--- program P_fl_2 (robot KUKA KR 16 2) ---
  Suave(1)
  Establecer velocidad (1000.0 mm/s)
  Est. Ref.: Frame 2
  Est. herr: Plumon_ensamble
  Mostrar Plumon_ensamble
  MoveJ 1 to (150.76, 185.35, 20) mm, rotated rx -180 ry 0 rz -39.83 deg; joints [47.982, -66.548, 70.781, -0.863, 85.768, 48.043]
  MoveL 2 to (150.76, 185.35, 20) mm, rotated rx -180 ry 0 rz -39.83 deg; joints [47.982, -66.548, 70.781, -0.863, 85.768, 48.043]
  MoveL 3 to (150.76, 185.35, 0) mm, rotated rx -180 ry 0 rz -39.83 deg; joints [47.968, -66.304, 72.161, -0.865, 84.143, 48.053]
  MoveL 4 to (150.76, 185.35, 0) mm, rotated rx -180 ry 0 rz -39.83 deg; joints [47.968, -66.304, 72.161, -0.865, 84.143, 48.053]
  Establecer velocidad (50.0 mm/s)
  MoveL 5 to (150.39, 185.32, 0) mm, rotated rx 180 ry 0 rz -39.83 deg; joints [47.95, -66.305, 72.163, -0.865, 84.143, 48.036]
  MoveL 6 to (150.03, 185.29, 0) mm, rotated rx 180 ry 0 rz -39.83 deg; joints [47.933, -66.307, 72.164, -0.865, 84.143, 48.018]
  MoveL 7 to (149.66, 185.26, 0) mm, rotated rx 180 ry 0 rz -39.83 deg; joints [47.915, -66.308, 72.165, -0.865, 84.142, 48]
  MoveL 8 to (149.29, 185.23, 0) mm, rotated rx 180 ry 0 rz -39.83 deg; joints [47.898, -66.309, 72.166, -0.865, 84.142, 47.983]
  MoveL 9 to (148.29, 185.2, 0) mm, rotated rx 180 ry 0 rz -39.83 deg; joints [47.85, -66.309, 72.165, -0.865, 84.143, 47.935]
  MoveL 10 to (147.29, 185.19, 0) mm, rotated rx 180 ry 0 rz -39.83 deg; joints [47.802, -66.306, 72.159, -0.865, 84.144, 47.887]
  MoveL 11 to (146.29, 185.21, 0) mm, rotated rx -180 ry 0 rz -39.83 deg; joints [47.754, -66.301, 72.151, -0.865, 84.147, 47.839]
  MoveL 12 to (145.28, 185.23, 0) mm, rotated rx -180 ry 0 rz -39.83 deg; joints [47.706, -66.295, 72.142, -0.865, 84.15, 47.791]
  MoveL 13 to (144.05, 185.27, 0) mm, rotated rx 180 ry 0 rz -39.83 deg; joints [47.647, -66.288, 72.129, -0.865, 84.154, 47.732]
  MoveL 14 to (142.82, 185.33, 0) mm, rotated rx -180 ry 0 rz -39.83 deg; joints [47.588, -66.278, 72.115, -0.865, 84.158, 47.673]
  MoveL 15 to (141.59, 185.42, 0) mm, rotated rx 180 ry 0 rz -39.83 deg; joints [47.53, -66.266, 72.096, -0.865, 84.164, 47.614]
  MoveL 16 to (140.37, 185.55, 0) mm, rotated rx -180 ry 0 rz -39.83 deg; joints [47.472, -66.25, 72.072, -0.865, 84.172, 47.556]
  MoveL 17 to (139.51, 185.68, 0) mm, rotated rx 180 ry 0 rz -39.83 deg; joints [47.431, -66.235, 72.05, -0.865, 84.178, 47.515]
  MoveL 18 to (138.64, 185.84, 0) mm, rotated rx 180 ry 0 rz -39.83 deg; joints [47.39, -66.219, 72.025, -0.865, 84.186, 47.474]
  MoveL 19 to (137.78, 186.01, 0) mm, rotated rx 180 ry 0 rz -39.83 deg; joints [47.349, -66.2, 71.997, -0.865, 84.194, 47.433]
  MoveL 20 to (136.93, 186.2, 0) mm, rotated rx 180 ry 0 rz -39.83 deg; joints [47.308, -66.18, 71.968, -0.865, 84.202, 47.393]
  MoveL 21 to (135.83, 186.46, 0) mm, rotated rx 180 ry 0 rz -39.83 deg; joints [47.257, -66.153, 71.929, -0.865, 84.214, 47.34]
  MoveL 22 to (134.73, 186.74, 0) mm, rotated rx 180 ry 0 rz -39.83 deg; joints [47.205, -66.125, 71.887, -0.865, 84.227, 47.289]
  MoveL 23 to (133.64, 187.03, 0) mm, rotated rx -180 ry 0 rz -39.83 deg; joints [47.154, -66.095, 71.843, -0.865, 84.24, 47.237]
  MoveL 24 to (132.56, 187.35, 0) mm, rotated rx 180 ry 0 rz -39.83 deg; joints [47.103, -66.063, 71.796, -0.865, 84.254, 47.186]
  MoveL 25 to (131.68, 187.63, 0) mm, rotated rx 180 ry 0 rz -39.83 deg; joints [47.062, -66.035, 71.756, -0.865, 84.266, 47.145]
  MoveL 26 to (130.81, 187.93, 0) mm, rotated rx -180 ry 0 rz -39.83 deg; joints [47.021, -66.005, 71.712, -0.865, 84.279, 47.104]
  MoveL 27 to (129.95, 188.26, 0) mm, rotated rx 180 ry 0 rz -39.83 deg; joints [46.981, -65.972, 71.665, -0.865, 84.293, 47.063]
  MoveL 28 to (129.1, 188.62, 0) mm, rotated rx -180 ry 0 rz -39.83 deg; joints [46.941, -65.937, 71.614, -0.865, 84.308, 47.024]
  MoveL 29 to (128.38, 188.97, 0) mm, rotated rx 180 ry 0 rz -39.83 deg; joints [46.908, -65.904, 71.566, -0.865, 84.322, 46.99]
  MoveL 30 to (127.67, 189.34, 0) mm, rotated rx 180 ry 0 rz -39.83 deg; joints [46.875, -65.868, 71.515, -0.865, 84.338, 46.957]
  MoveL 31 to (126.97, 189.74, 0) mm, rotated rx 180 ry 0 rz -39.83 deg; joints [46.843, -65.83, 71.46, -0.865, 84.354, 46.925]
  MoveL 32 to (126.29, 190.17, 0) mm, rotated rx -180 ry 0 rz -39.83 deg; joints [46.812, -65.79, 71.401, -0.865, 84.371, 46.893]
  MoveL 33 to (125.71, 190.58, 0) mm, rotated rx 180 ry 0 rz -39.83 deg; joints [46.785, -65.752, 71.347, -0.865, 84.388, 46.866]
  MoveL 34 to (125.14, 191, 0) mm, rotated rx -180 ry 0 rz -39.83 deg; joints [46.76, -65.713, 71.29, -0.865, 84.405, 46.84]
  MoveL 35 to (124.6, 191.45, 0) mm, rotated rx -180 ry 0 rz -39.83 deg; joints [46.735, -65.671, 71.23, -0.865, 84.422, 46.816]
  MoveL 36 to (124.08, 191.93, 0) mm, rotated rx -180 ry 0 rz -39.83 deg; joints [46.712, -65.627, 71.167, -0.864, 84.441, 46.792]
  MoveL 37 to (123.59, 192.43, 0) mm, rotated rx 180 ry 0 rz -39.83 deg; joints [46.69, -65.582, 71.102, -0.864, 84.461, 46.77]
  MoveL 38 to (123.13, 192.95, 0) mm, rotated rx 180 ry 0 rz -39.83 deg; joints [46.669, -65.534, 71.034, -0.864, 84.481, 46.749]
  MoveL 39 to (122.67, 193.48, 0) mm, rotated rx -180 ry 0 rz -39.83 deg; joints [46.649, -65.486, 70.964, -0.864, 84.502, 46.729]
  MoveL 40 to (122.23, 194.03, 0) mm, rotated rx -180 ry 0 rz -39.83 deg; joints [46.63, -65.436, 70.893, -0.864, 84.523, 46.709]
  MoveL 41 to (121.75, 194.65, 0) mm, rotated rx 180 ry 0 rz -39.83 deg; joints [46.609, -65.38, 70.812, -0.864, 84.548, 46.688]
  MoveL 42 to (121.29, 195.28, 0) mm, rotated rx -180 ry 0 rz -39.83 deg; joints [46.589, -65.323, 70.73, -0.864, 84.572, 46.667]
  MoveL 43 to (120.86, 195.94, 0) mm, rotated rx 180 ry 0 rz -39.83 deg; joints [46.571, -65.264, 70.645, -0.864, 84.598, 46.649]
  MoveL 44 to (120.5, 196.62, 0) mm, rotated rx -180 ry 0 rz -39.83 deg; joints [46.556, -65.203, 70.558, -0.864, 84.624, 46.633]
  MoveL 45 to (120.13, 197.53, 0) mm, rotated rx 180 ry 0 rz -39.83 deg; joints [46.541, -65.121, 70.441, -0.864, 84.66, 46.618]
  MoveL 46 to (119.85, 198.49, 0) mm, rotated rx 180 ry 0 rz -39.83 deg; joints [46.531, -65.037, 70.32, -0.864, 84.696, 46.607]
  MoveL 47 to (119.64, 199.47, 0) mm, rotated rx 180 ry 0 rz -39.83 deg; joints [46.523, -64.95, 70.195, -0.864, 84.734, 46.599]
  MoveL 48 to (119.45, 200.46, 0) mm, rotated rx 180 ry 0 rz -39.83 deg; joints [46.518, -64.863, 70.07, -0.864, 84.772, 46.593]
  Establecer velocidad (1000.0 mm/s)
  MoveL 49 to (119.45, 200.46, 0) mm, rotated rx 180 ry 0 rz -39.83 deg; joints [46.518, -64.863, 70.07, -0.864, 84.772, 46.593]
  MoveL 50 to (119.45, 200.46, 20) mm, rotated rx 180 ry 0 rz -39.83 deg; joints [46.532, -65.091, 68.674, -0.862, 86.395, 46.583]
  Establecer velocidad (1000.0 mm/s)
  MoveL 51 to (146.94, 188.19, 20) mm, rotated rx 180 ry 0 rz -39.83 deg; joints [47.806, -66.288, 70.409, -0.863, 85.877, 47.864]
  MoveL 52 to (146.94, 188.19, 0) mm, rotated rx 180 ry 0 rz -39.83 deg; joints [47.791, -66.046, 71.792, -0.865, 84.252, 47.875]
  MoveL 53 to (146.94, 188.19, 0) mm, rotated rx 180 ry 0 rz -39.83 deg; joints [47.791, -66.046, 71.792, -0.865, 84.252, 47.875]
  Establecer velocidad (50.0 mm/s)
  MoveL 54 to (147.05, 187.92, 0) mm, rotated rx -180 ry 0 rz -39.83 deg; joints [47.796, -66.07, 71.826, -0.865, 84.242, 47.879]
  MoveL 55 to (147.17, 187.65, 0) mm, rotated rx 180 ry 0 rz -39.83 deg; joints [47.801, -66.094, 71.86, -0.865, 84.232, 47.885]
  MoveL 56 to (147.31, 187.4, 0) mm, rotated rx 180 ry 0 rz -39.83 deg; joints [47.807, -66.116, 71.891, -0.865, 84.223, 47.891]
  MoveL 57 to (147.47, 187.17, 0) mm, rotated rx 180 ry 0 rz -39.83 deg; joints [47.814, -66.136, 71.92, -0.865, 84.215, 47.898]
  MoveL 58 to (147.77, 186.91, 0) mm, rotated rx 180 ry 0 rz -39.83 deg; joints [47.828, -66.159, 71.953, -0.865, 84.205, 47.912]
  MoveL 59 to (148.12, 186.7, 0) mm, rotated rx 180 ry 0 rz -39.83 deg; joints [47.844, -66.179, 71.981, -0.865, 84.197, 47.929]
  MoveL 60 to (148.5, 186.52, 0) mm, rotated rx 180 ry 0 rz -39.83 deg; joints [47.862, -66.195, 72.005, -0.865, 84.189, 47.946]
  MoveL 61 to (148.88, 186.35, 0) mm, rotated rx -180 ry 0 rz -39.83 deg; joints [47.88, -66.211, 72.028, -0.865, 84.183, 47.965]
  MoveL 62 to (149.37, 186.12, 0) mm, rotated rx 180 ry 0 rz -39.83 deg; joints [47.903, -66.233, 72.059, -0.865, 84.173, 47.988]
  MoveL 63 to (149.85, 185.87, 0) mm, rotated rx 180 ry 0 rz -39.83 deg; joints [47.925, -66.256, 72.092, -0.865, 84.164, 48.01]
  MoveL 64 to (150.3, 185.61, 0) mm, rotated rx 180 ry 0 rz -39.83 deg; joints [47.947, -66.28, 72.126, -0.865, 84.154, 48.032]
  MoveL 65 to (150.76, 185.35, 0) mm, rotated rx -180 ry 0 rz -39.83 deg; joints [47.968, -66.304, 72.161, -0.865, 84.143, 48.053]
  Establecer velocidad (1000.0 mm/s)
  MoveL 66 to (150.76, 185.35, 0) mm, rotated rx -180 ry 0 rz -39.83 deg; joints [47.968, -66.304, 72.161, -0.865, 84.143, 48.053]
  MoveL 67 to (150.76, 185.35, 20) mm, rotated rx -180 ry 0 rz -39.83 deg; joints [47.982, -66.548, 70.781, -0.863, 85.768, 48.043]
  Establecer velocidad (1000.0 mm/s)
  MoveL 68 to (146.94, 188.19, 20) mm, rotated rx 180 ry 0 rz -39.83 deg; joints [47.806, -66.288, 70.409, -0.863, 85.877, 47.864]
  MoveL 69 to (146.94, 188.19, 0) mm, rotated rx 180 ry 0 rz -39.83 deg; joints [47.791, -66.046, 71.792, -0.865, 84.252, 47.875]
  MoveL 70 to (146.94, 188.19, 0) mm, rotated rx 180 ry 0 rz -39.83 deg; joints [47.791, -66.046, 71.792, -0.865, 84.252, 47.875]
  Establecer velocidad (50.0 mm/s)
  MoveL 71 to (147.49, 188.32, 0) mm, rotated rx -180 ry 0 rz -39.83 deg; joints [47.817, -66.037, 71.779, -0.865, 84.256, 47.901]
  MoveL 72 to (148.03, 188.44, 0) mm, rotated rx -180 ry 0 rz -39.83 deg; joints [47.844, -66.029, 71.768, -0.865, 84.259, 47.927]
  MoveL 73 to (148.58, 188.53, 0) mm, rotated rx -180 ry 0 rz -39.83 deg; joints [47.87, -66.022, 71.76, -0.865, 84.261, 47.953]
  MoveL 74 to (149.12, 188.6, 0) mm, rotated rx 180 ry 0 rz -39.83 deg; joints [47.896, -66.018, 71.755, -0.865, 84.263, 47.979]
  MoveL 75 to (149.7, 188.63, 0) mm, rotated rx 180 ry 0 rz -39.83 deg; joints [47.923, -66.018, 71.755, -0.865, 84.262, 48.007]
  MoveL 76 to (150.27, 188.63, 0) mm, rotated rx -180 ry 0 rz -39.83 deg; joints [47.951, -66.019, 71.758, -0.865, 84.261, 48.034]
  MoveL 77 to (150.85, 188.62, 0) mm, rotated rx 180 ry 0 rz -39.83 deg; joints [47.978, -66.022, 71.762, -0.865, 84.26, 48.062]
  MoveL 78 to (151.43, 188.62, 0) mm, rotated rx 180 ry 0 rz -39.83 deg; joints [48.006, -66.024, 71.766, -0.865, 84.259, 48.089]
  MoveL 79 to (152.23, 188.66, 0) mm, rotated rx 180 ry 0 rz -39.83 deg; joints [48.044, -66.023, 71.766, -0.865, 84.259, 48.128]
  MoveL 80 to (153.02, 188.73, 0) mm, rotated rx 180 ry 0 rz -39.83 deg; joints [48.082, -66.019, 71.761, -0.865, 84.26, 48.166]
  MoveL 81 to (153.81, 188.83, 0) mm, rotated rx 180 ry 0 rz -39.83 deg; joints [48.12, -66.012, 71.753, -0.865, 84.262, 48.204]
  MoveL 82 to (154.6, 188.96, 0) mm, rotated rx 180 ry 0 rz -39.83 deg; joints [48.158, -66.004, 71.742, -0.865, 84.265, 48.241]
  MoveL 83 to (155.12, 189.06, 0) mm, rotated rx 180 ry 0 rz -39.83 deg; joints [48.183, -65.997, 71.733, -0.865, 84.268, 48.266]
  MoveL 84 to (155.65, 189.15, 0) mm, rotated rx 180 ry 0 rz -39.83 deg; joints [48.208, -65.99, 71.723, -0.865, 84.271, 48.291]
  MoveL 85 to (156.18, 189.25, 0) mm, rotated rx 180 ry 0 rz -39.83 deg; joints [48.234, -65.983, 71.714, -0.865, 84.273, 48.317]
  MoveL 86 to (156.72, 189.34, 0) mm, rotated rx 180 ry 0 rz -39.83 deg; joints [48.26, -65.976, 71.706, -0.865, 84.276, 48.343]
  MoveL 87 to (157.41, 189.46, 0) mm, rotated rx 180 ry 0 rz -39.83 deg; joints [48.293, -65.969, 71.696, -0.865, 84.278, 48.376]
  MoveL 88 to (158.09, 189.6, 0) mm, rotated rx 180 ry 0 rz -39.83 deg; joints [48.326, -65.958, 71.682, -0.865, 84.282, 48.409]
  MoveL 89 to (158.73, 189.82, 0) mm, rotated rx 180 ry 0 rz -39.83 deg; joints [48.356, -65.941, 71.658, -0.865, 84.289, 48.439]
  MoveL 90 to (159.28, 190.16, 0) mm, rotated rx 180 ry 0 rz -39.83 deg; joints [48.383, -65.913, 71.619, -0.865, 84.301, 48.466]
  MoveL 91 to (159.48, 190.35, 0) mm, rotated rx 180 ry 0 rz -39.83 deg; joints [48.393, -65.897, 71.597, -0.865, 84.307, 48.475]
  MoveL 92 to (159.66, 190.56, 0) mm, rotated rx 180 ry 0 rz -39.83 deg; joints [48.402, -65.879, 71.572, -0.865, 84.314, 48.484]
  MoveL 93 to (159.83, 190.78, 0) mm, rotated rx 180 ry 0 rz -39.83 deg; joints [48.41, -65.86, 71.545, -0.865, 84.322, 48.493]
  MoveL 94 to (160, 191.02, 0) mm, rotated rx 180 ry 0 rz -39.83 deg; joints [48.419, -65.84, 71.517, -0.865, 84.331, 48.501]
  MoveL 95 to (160, 191.02, 0) mm, rotated rx 180 ry 0 rz -39.83 deg; joints [48.419, -65.84, 71.517, -0.865, 84.331, 48.501]
  MoveL 96 to (159.66, 191.06, 0) mm, rotated rx 180 ry 0 rz -39.83 deg; joints [48.403, -65.836, 71.51, -0.865, 84.333, 48.485]
  MoveL 97 to (159.32, 191.11, 0) mm, rotated rx 180 ry 0 rz -39.83 deg; joints [48.387, -65.831, 71.502, -0.865, 84.335, 48.469]
  MoveL 98 to (158.98, 191.16, 0) mm, rotated rx 180 ry 0 rz -39.83 deg; joints [48.371, -65.825, 71.494, -0.865, 84.337, 48.453]
  MoveL 99 to (158.65, 191.22, 0) mm, rotated rx 180 ry 0 rz -39.83 deg; joints [48.355, -65.819, 71.486, -0.865, 84.34, 48.437]
  MoveL 100 to (158.29, 191.29, 0) mm, rotated rx 180 ry 0 rz -39.83 deg; joints [48.338, -65.812, 71.475, -0.865, 84.343, 48.42]
  MoveL 101 to (157.93, 191.38, 0) mm, rotated rx 180 ry 0 rz -39.83 deg; joints [48.321, -65.804, 71.463, -0.865, 84.347, 48.403]
  MoveL 102 to (157.58, 191.47, 0) mm, rotated rx 180 ry 0 rz -39.83 deg; joints [48.304, -65.795, 71.45, -0.865, 84.351, 48.386]
  MoveL 103 to (157.22, 191.58, 0) mm, rotated rx 180 ry 0 rz -39.83 deg; joints [48.287, -65.785, 71.435, -0.865, 84.355, 48.369]
  MoveL 104 to (157.01, 191.65, 0) mm, rotated rx 180 ry 0 rz -39.83 deg; joints [48.277, -65.778, 71.425, -0.865, 84.358, 48.359]
  MoveL 105 to (156.8, 191.73, 0) mm, rotated rx 180 ry 0 rz -39.83 deg; joints [48.267, -65.77, 71.414, -0.865, 84.362, 48.349]
  MoveL 106 to (156.6, 191.84, 0) mm, rotated rx 180 ry 0 rz -39.83 deg; joints [48.258, -65.761, 71.4, -0.865, 84.366, 48.34]
  MoveL 107 to (156.43, 191.97, 0) mm, rotated rx 180 ry 0 rz -39.83 deg; joints [48.25, -65.749, 71.382, -0.865, 84.371, 48.332]
  MoveL 108 to (156.31, 192.1, 0) mm, rotated rx -180 ry 0 rz -39.83 deg; joints [48.245, -65.737, 71.366, -0.865, 84.376, 48.326]
  MoveL 109 to (156.21, 192.24, 0) mm, rotated rx 180 ry 0 rz -39.83 deg; joints [48.24, -65.725, 71.348, -0.865, 84.381, 48.322]
  MoveL 110 to (156.14, 192.4, 0) mm, rotated rx 180 ry 0 rz -39.83 deg; joints [48.237, -65.711, 71.328, -0.865, 84.387, 48.318]
  MoveL 111 to (156.09, 192.57, 0) mm, rotated rx 180 ry 0 rz -39.83 deg; joints [48.235, -65.696, 71.308, -0.865, 84.393, 48.316]
  MoveL 112 to (156.07, 192.68, 0) mm, rotated rx 180 ry 0 rz -39.83 deg; joints [48.234, -65.687, 71.294, -0.865, 84.397, 48.316]
  MoveL 113 to (156.07, 192.79, 0) mm, rotated rx 180 ry 0 rz -39.83 deg; joints [48.234, -65.677, 71.28, -0.865, 84.402, 48.315]
  MoveL 114 to (156.07, 192.9, 0) mm, rotated rx 180 ry 0 rz -39.83 deg; joints [48.235, -65.667, 71.266, -0.865, 84.406, 48.316]
  MoveL 115 to (156.07, 193.02, 0) mm, rotated rx -180 ry 0 rz -39.83 deg; joints [48.235, -65.657, 71.252, -0.865, 84.41, 48.316]
  MoveL 116 to (156.07, 193.02, 0) mm, rotated rx -180 ry 0 rz -39.83 deg; joints [48.235, -65.657, 71.252, -0.865, 84.41, 48.316]
  MoveL 117 to (156.36, 193.11, 0) mm, rotated rx 180 ry 0 rz -39.83 deg; joints [48.249, -65.65, 71.243, -0.865, 84.413, 48.33]
  MoveL 118 to (156.65, 193.19, 0) mm, rotated rx 180 ry 0 rz -39.83 deg; joints [48.262, -65.644, 71.234, -0.865, 84.415, 48.343]
  MoveL 119 to (156.94, 193.27, 0) mm, rotated rx -180 ry 0 rz -39.83 deg; joints [48.276, -65.638, 71.225, -0.865, 84.418, 48.357]
  MoveL 120 to (157.22, 193.35, 0) mm, rotated rx 180 ry 0 rz -39.83 deg; joints [48.29, -65.632, 71.217, -0.865, 84.42, 48.371]
  MoveL 121 to (157.72, 193.46, 0) mm, rotated rx -180 ry 0 rz -39.83 deg; joints [48.314, -65.624, 71.206, -0.865, 84.423, 48.395]
  MoveL 122 to (158.22, 193.55, 0) mm, rotated rx 180 ry 0 rz -39.83 deg; joints [48.338, -65.617, 71.197, -0.865, 84.426, 48.419]
  MoveL 123 to (158.72, 193.64, 0) mm, rotated rx 180 ry 0 rz -39.83 deg; joints [48.362, -65.611, 71.189, -0.865, 84.428, 48.443]
  MoveL 124 to (159.22, 193.73, 0) mm, rotated rx -180 ry 0 rz -39.83 deg; joints [48.386, -65.604, 71.18, -0.865, 84.431, 48.467]
  MoveL 125 to (159.66, 193.82, 0) mm, rotated rx 180 ry 0 rz -39.83 deg; joints [48.407, -65.597, 71.171, -0.865, 84.433, 48.487]
  MoveL 126 to (160.09, 193.92, 0) mm, rotated rx 180 ry 0 rz -39.83 deg; joints [48.427, -65.59, 71.161, -0.865, 84.436, 48.508]
  MoveL 127 to (160.52, 194.02, 0) mm, rotated rx -180 ry 0 rz -39.83 deg; joints [48.448, -65.582, 71.151, -0.865, 84.439, 48.528]
  MoveL 128 to (160.95, 194.13, 0) mm, rotated rx -180 ry 0 rz -39.83 deg; joints [48.468, -65.573, 71.139, -0.865, 84.442, 48.549]
  MoveL 129 to (161.5, 194.28, 0) mm, rotated rx 180 ry 0 rz -39.83 deg; joints [48.495, -65.562, 71.123, -0.865, 84.447, 48.575]
  MoveL 130 to (162.04, 194.44, 0) mm, rotated rx 180 ry 0 rz -39.83 deg; joints [48.521, -65.55, 71.106, -0.865, 84.452, 48.601]
  MoveL 131 to (162.59, 194.6, 0) mm, rotated rx 180 ry 0 rz -39.83 deg; joints [48.547, -65.537, 71.089, -0.865, 84.457, 48.627]
  MoveL 132 to (163.13, 194.77, 0) mm, rotated rx -180 ry 0 rz -39.83 deg; joints [48.573, -65.523, 71.071, -0.865, 84.462, 48.653]
  MoveL 133 to (163.88, 195.01, 0) mm, rotated rx 180 ry 0 rz -39.83 deg; joints [48.609, -65.504, 71.044, -0.865, 84.47, 48.689]
  MoveL 134 to (164.62, 195.28, 0) mm, rotated rx 180 ry 0 rz -39.83 deg; joints [48.644, -65.482, 71.013, -0.865, 84.479, 48.724]
  MoveL 135 to (165.34, 195.59, 0) mm, rotated rx -180 ry 0 rz -39.83 deg; joints [48.679, -65.457, 70.978, -0.865, 84.489, 48.759]
  MoveL 136 to (166.05, 195.95, 0) mm, rotated rx 180 ry 0 rz -39.83 deg; joints [48.713, -65.427, 70.937, -0.865, 84.502, 48.793]
  MoveL 137 to (166.39, 196.15, 0) mm, rotated rx -180 ry 0 rz -39.83 deg; joints [48.73, -65.41, 70.913, -0.865, 84.509, 48.809]
  MoveL 138 to (166.71, 196.38, 0) mm, rotated rx -180 ry 0 rz -39.83 deg; joints [48.745, -65.391, 70.887, -0.865, 84.517, 48.825]
  MoveL 139 to (167.01, 196.63, 0) mm, rotated rx -180 ry 0 rz -39.83 deg; joints [48.759, -65.37, 70.857, -0.864, 84.525, 48.839]
  MoveL 140 to (167.26, 196.91, 0) mm, rotated rx 180 ry 0 rz -39.83 deg; joints [48.772, -65.346, 70.823, -0.864, 84.536, 48.851]
  MoveL 141 to (167.41, 197.13, 0) mm, rotated rx 180 ry 0 rz -39.83 deg; joints [48.779, -65.327, 70.797, -0.864, 84.543, 48.858]
  MoveL 142 to (167.55, 197.36, 0) mm, rotated rx 180 ry 0 rz -39.83 deg; joints [48.786, -65.308, 70.769, -0.864, 84.552, 48.865]
  MoveL 143 to (167.67, 197.6, 0) mm, rotated rx 180 ry 0 rz -39.83 deg; joints [48.792, -65.287, 70.739, -0.864, 84.561, 48.871]
  MoveL 144 to (167.79, 197.85, 0) mm, rotated rx -180 ry 0 rz -39.83 deg; joints [48.798, -65.266, 70.709, -0.864, 84.569, 48.877]
  MoveL 145 to (167.79, 197.85, 0) mm, rotated rx -180 ry 0 rz -39.83 deg; joints [48.798, -65.266, 70.709, -0.864, 84.569, 48.877]
  MoveL 146 to (167.56, 197.78, 0) mm, rotated rx -180 ry 0 rz -39.83 deg; joints [48.787, -65.271, 70.717, -0.864, 84.567, 48.865]
  MoveL 147 to (167.32, 197.71, 0) mm, rotated rx 180 ry 0 rz -39.83 deg; joints [48.776, -65.277, 70.724, -0.864, 84.565, 48.854]
  MoveL 148 to (167.09, 197.65, 0) mm, rotated rx -180 ry 0 rz -39.83 deg; joints [48.764, -65.281, 70.731, -0.864, 84.563, 48.843]
  MoveL 149 to (166.85, 197.6, 0) mm, rotated rx 180 ry 0 rz -39.83 deg; joints [48.753, -65.286, 70.737, -0.864, 84.561, 48.832]
  MoveL 150 to (166.29, 197.5, 0) mm, rotated rx 180 ry 0 rz -39.83 deg; joints [48.727, -65.293, 70.746, -0.864, 84.559, 48.805]
  MoveL 151 to (165.73, 197.46, 0) mm, rotated rx -180 ry 0 rz -39.83 deg; joints [48.7, -65.295, 70.749, -0.864, 84.558, 48.779]
  MoveL 152 to (165.17, 197.48, 0) mm, rotated rx 180 ry 0 rz -39.83 deg; joints [48.673, -65.292, 70.744, -0.864, 84.56, 48.752]
  MoveL 153 to (164.61, 197.57, 0) mm, rotated rx 180 ry 0 rz -39.83 deg; joints [48.647, -65.283, 70.73, -0.864, 84.564, 48.726]
  MoveL 154 to (164.15, 197.71, 0) mm, rotated rx 180 ry 0 rz -39.83 deg; joints [48.625, -65.27, 70.711, -0.864, 84.57, 48.704]
  MoveL 155 to (163.69, 197.89, 0) mm, rotated rx -180 ry 0 rz -39.83 deg; joints [48.604, -65.254, 70.686, -0.864, 84.577, 48.682]
  MoveL 156 to (163.25, 198.1, 0) mm, rotated rx -180 ry 0 rz -39.83 deg; joints [48.583, -65.234, 70.658, -0.864, 84.586, 48.661]
  MoveL 157 to (162.81, 198.33, 0) mm, rotated rx -180 ry 0 rz -39.83 deg; joints [48.562, -65.214, 70.629, -0.864, 84.595, 48.641]
  MoveL 158 to (162.81, 198.33, 0) mm, rotated rx -180 ry 0 rz -39.83 deg; joints [48.562, -65.214, 70.629, -0.864, 84.595, 48.641]
  MoveL 159 to (164.35, 199.04, 0) mm, rotated rx 180 ry 0 rz -39.83 deg; joints [48.637, -65.155, 70.547, -0.864, 84.619, 48.715]
  MoveL 160 to (165.89, 199.78, 0) mm, rotated rx 180 ry 0 rz -39.83 deg; joints [48.71, -65.094, 70.461, -0.864, 84.644, 48.788]
  MoveL 161 to (167.39, 200.56, 0) mm, rotated rx 180 ry 0 rz -39.83 deg; joints [48.782, -65.029, 70.37, -0.864, 84.672, 48.859]
  MoveL 162 to (168.86, 201.41, 0) mm, rotated rx 180 ry 0 rz -39.83 deg; joints [48.852, -64.958, 70.271, -0.864, 84.701, 48.929]
  MoveL 163 to (170.25, 202.31, 0) mm, rotated rx -180 ry 0 rz -39.83 deg; joints [48.919, -64.882, 70.163, -0.864, 84.734, 48.995]
  MoveL 164 to (171.6, 203.28, 0) mm, rotated rx 180 ry 0 rz -39.83 deg; joints [48.984, -64.8, 70.047, -0.864, 84.769, 49.06]
  MoveL 165 to (172.93, 204.29, 0) mm, rotated rx 180 ry 0 rz -39.83 deg; joints [49.047, -64.714, 69.925, -0.864, 84.805, 49.123]
  MoveL 166 to (174.24, 205.32, 0) mm, rotated rx 180 ry 0 rz -39.83 deg; joints [49.11, -64.626, 69.801, -0.864, 84.843, 49.185]
  MoveL 167 to (174.24, 205.32, 0) mm, rotated rx 180 ry 0 rz -39.83 deg; joints [49.11, -64.626, 69.801, -0.864, 84.843, 49.185]
  MoveL 168 to (173.58, 205.32, 0) mm, rotated rx 180 ry 0 rz -39.83 deg; joints [49.079, -64.625, 69.798, -0.864, 84.844, 49.154]
  MoveL 169 to (172.92, 205.32, 0) mm, rotated rx 180 ry 0 rz -39.83 deg; joints [49.048, -64.624, 69.796, -0.864, 84.845, 49.123]
  MoveL 170 to (172.25, 205.3, 0) mm, rotated rx -180 ry 0 rz -39.83 deg; joints [49.017, -64.625, 69.796, -0.864, 84.845, 49.091]
  MoveL 171 to (171.57, 205.27, 0) mm, rotated rx -180 ry 0 rz -39.83 deg; joints [48.985, -64.627, 69.798, -0.864, 84.844, 49.059]
  MoveL 172 to (171.05, 205.23, 0) mm, rotated rx 180 ry 0 rz -39.83 deg; joints [48.96, -64.629, 69.801, -0.864, 84.844, 49.034]
  MoveL 173 to (170.52, 205.22, 0) mm, rotated rx 180 ry 0 rz -39.83 deg; joints [48.935, -64.629, 69.8, -0.864, 84.844, 49.01]
  MoveL 174 to (170.02, 205.26, 0) mm, rotated rx 180 ry 0 rz -39.83 deg; joints [48.911, -64.624, 69.793, -0.864, 84.846, 48.986]
  MoveL 175 to (169.55, 205.41, 0) mm, rotated rx -180 ry 0 rz -39.83 deg; joints [48.89, -64.611, 69.772, -0.864, 84.852, 48.964]
  MoveL 176 to (169.36, 205.51, 0) mm, rotated rx -180 ry 0 rz -39.83 deg; joints [48.881, -64.601, 69.759, -0.864, 84.857, 48.955]
  MoveL 177 to (169.18, 205.64, 0) mm, rotated rx -180 ry 0 rz -39.83 deg; joints [48.872, -64.59, 69.742, -0.864, 84.862, 48.946]
  MoveL 178 to (169, 205.78, 0) mm, rotated rx -180 ry 0 rz -39.83 deg; joints [48.864, -64.578, 69.724, -0.864, 84.867, 48.938]
  MoveL 179 to (168.82, 205.92, 0) mm, rotated rx 180 ry 0 rz -39.83 deg; joints [48.855, -64.565, 69.705, -0.864, 84.873, 48.93]
  MoveL 180 to (168.82, 205.92, 0) mm, rotated rx 180 ry 0 rz -39.83 deg; joints [48.855, -64.565, 69.705, -0.864, 84.873, 48.93]
  MoveL 181 to (169.99, 206.54, 0) mm, rotated rx 180 ry 0 rz -39.83 deg; joints [48.911, -64.513, 69.632, -0.864, 84.895, 48.985]
  MoveL 182 to (171.15, 207.17, 0) mm, rotated rx 180 ry 0 rz -39.83 deg; joints [48.966, -64.459, 69.557, -0.864, 84.918, 49.04]
  MoveL 183 to (172.27, 207.85, 0) mm, rotated rx 180 ry 0 rz -39.83 deg; joints [49.02, -64.402, 69.476, -0.864, 84.943, 49.093]
  MoveL 184 to (173.36, 208.58, 0) mm, rotated rx 180 ry 0 rz -39.83 deg; joints [49.072, -64.34, 69.387, -0.864, 84.97, 49.144]
  MoveL 185 to (174.61, 209.58, 0) mm, rotated rx 180 ry 0 rz -39.83 deg; joints [49.131, -64.254, 69.265, -0.864, 85.007, 49.204]
  MoveL 186 to (175.8, 210.66, 0) mm, rotated rx 180 ry 0 rz -39.83 deg; joints [49.188, -64.161, 69.132, -0.864, 85.048, 49.259]
  MoveL 187 to (176.94, 211.81, 0) mm, rotated rx 180 ry 0 rz -39.83 deg; joints [49.242, -64.062, 68.99, -0.864, 85.091, 49.313]
  MoveL 188 to (178.06, 212.98, 0) mm, rotated rx -180 ry 0 rz -39.83 deg; joints [49.296, -63.96, 68.844, -0.864, 85.136, 49.366]
  MoveL 189 to (178.06, 212.98, 0) mm, rotated rx -180 ry 0 rz -39.83 deg; joints [49.296, -63.96, 68.844, -0.864, 85.136, 49.366]
  MoveL 190 to (177.4, 212.99, 0) mm, rotated rx 180 ry 0 rz -39.83 deg; joints [49.265, -63.959, 68.842, -0.864, 85.137, 49.335]
  MoveL 191 to (176.74, 212.99, 0) mm, rotated rx 180 ry 0 rz -39.83 deg; joints [49.234, -63.958, 68.839, -0.864, 85.138, 49.304]
  MoveL 192 to (176.07, 212.99, 0) mm, rotated rx -180 ry 0 rz -39.83 deg; joints [49.203, -63.957, 68.837, -0.864, 85.139, 49.273]
  MoveL 193 to (175.4, 212.98, 0) mm, rotated rx -180 ry 0 rz -39.83 deg; joints [49.171, -63.957, 68.837, -0.864, 85.139, 49.241]
  MoveL 194 to (175.01, 212.97, 0) mm, rotated rx 180 ry 0 rz -39.83 deg; joints [49.153, -63.957, 68.836, -0.864, 85.139, 49.223]
  MoveL 195 to (174.62, 212.98, 0) mm, rotated rx 180 ry 0 rz -39.83 deg; joints [49.135, -63.956, 68.834, -0.864, 85.14, 49.205]
  MoveL 196 to (174.23, 213.01, 0) mm, rotated rx -180 ry 0 rz -39.83 deg; joints [49.117, -63.952, 68.828, -0.864, 85.142, 49.187]
  MoveL 197 to (173.87, 213.1, 0) mm, rotated rx -180 ry 0 rz -39.83 deg; joints [49.1, -63.944, 68.815, -0.864, 85.146, 49.17]
  MoveL 198 to (173.68, 213.17, 0) mm, rotated rx -180 ry 0 rz -39.83 deg; joints [49.091, -63.937, 68.806, -0.864, 85.149, 49.161]
  MoveL 199 to (173.5, 213.26, 0) mm, rotated rx 180 ry 0 rz -39.83 deg; joints [49.083, -63.93, 68.795, -0.864, 85.152, 49.153]
  MoveL 200 to (173.33, 213.35, 0) mm, rotated rx 180 ry 0 rz -39.83 deg; joints [49.075, -63.922, 68.782, -0.864, 85.156, 49.144]
  MoveL 201 to (173.15, 213.45, 0) mm, rotated rx 180 ry 0 rz -39.83 deg; joints [49.067, -63.913, 68.769, -0.864, 85.16, 49.136]
  MoveL 202 to (173.15, 213.45, 0) mm, rotated rx 180 ry 0 rz -39.83 deg; joints [49.067, -63.913, 68.769, -0.864, 85.16, 49.136]
  MoveL 203 to (174.19, 214.25, 0) mm, rotated rx 180 ry 0 rz -39.83 deg; joints [49.116, -63.844, 68.671, -0.864, 85.191, 49.185]
  MoveL 204 to (175.21, 215.06, 0) mm, rotated rx -180 ry 0 rz -39.83 deg; joints [49.164, -63.773, 68.57, -0.863, 85.222, 49.233]
  MoveL 205 to (176.21, 215.91, 0) mm, rotated rx 180 ry 0 rz -39.83 deg; joints [49.211, -63.7, 68.465, -0.863, 85.254, 49.28]
  MoveL 206 to (177.15, 216.8, 0) mm, rotated rx -180 ry 0 rz -39.83 deg; joints [49.256, -63.623, 68.354, -0.863, 85.289, 49.324]
  MoveL 207 to (178.22, 217.94, 0) mm, rotated rx 180 ry 0 rz -39.83 deg; joints [49.307, -63.523, 68.211, -0.863, 85.333, 49.374]
  MoveL 208 to (179.22, 219.15, 0) mm, rotated rx -180 ry 0 rz -39.83 deg; joints [49.354, -63.418, 68.058, -0.863, 85.381, 49.421]
  MoveL 209 to (180.18, 220.41, 0) mm, rotated rx 180 ry 0 rz -39.83 deg; joints [49.4, -63.308, 67.899, -0.863, 85.431, 49.466]
  MoveL 210 to (181.11, 221.68, 0) mm, rotated rx 180 ry 0 rz -39.83 deg; joints [49.444, -63.196, 67.738, -0.863, 85.481, 49.509]
  MoveL 211 to (181.11, 221.68, 0) mm, rotated rx 180 ry 0 rz -39.83 deg; joints [49.444, -63.196, 67.738, -0.863, 85.481, 49.509]
  MoveL 212 to (180.62, 221.61, 0) mm, rotated rx -180 ry 0 rz -39.83 deg; joints [49.421, -63.202, 67.745, -0.863, 85.479, 49.486]
  MoveL 213 to (180.12, 221.55, 0) mm, rotated rx 180 ry 0 rz -39.83 deg; joints [49.398, -63.207, 67.752, -0.863, 85.477, 49.463]
  MoveL 214 to (179.63, 221.49, 0) mm, rotated rx 180 ry 0 rz -39.83 deg; joints [49.375, -63.212, 67.758, -0.863, 85.475, 49.44]
  MoveL 215 to (179.13, 221.44, 0) mm, rotated rx -180 ry 0 rz -39.83 deg; joints [49.352, -63.216, 67.763, -0.863, 85.474, 49.417]
  MoveL 216 to (178.68, 221.41, 0) mm, rotated rx -180 ry 0 rz -39.83 deg; joints [49.331, -63.218, 67.766, -0.863, 85.473, 49.396]
  MoveL 217 to (178.23, 221.39, 0) mm, rotated rx 180 ry 0 rz -39.83 deg; joints [49.31, -63.219, 67.767, -0.863, 85.473, 49.375]
  MoveL 218 to (177.77, 221.39, 0) mm, rotated rx 180 ry 0 rz -39.83 deg; joints [49.288, -63.219, 67.766, -0.863, 85.473, 49.353]
  MoveL 219 to (177.31, 221.41, 0) mm, rotated rx 180 ry 0 rz -39.83 deg; joints [49.267, -63.216, 67.762, -0.863, 85.475, 49.332]
  MoveL 220 to (177.01, 221.44, 0) mm, rotated rx 180 ry 0 rz -39.83 deg; joints [49.253, -63.213, 67.757, -0.863, 85.476, 49.318]
  MoveL 221 to (176.71, 221.49, 0) mm, rotated rx 180 ry 0 rz -39.83 deg; joints [49.239, -63.208, 67.749, -0.863, 85.478, 49.304]
  MoveL 222 to (176.43, 221.57, 0) mm, rotated rx -180 ry 0 rz -39.83 deg; joints [49.226, -63.201, 67.738, -0.863, 85.482, 49.291]
  MoveL 223 to (176.18, 221.7, 0) mm, rotated rx 180 ry 0 rz -39.83 deg; joints [49.214, -63.189, 67.721, -0.863, 85.488, 49.279]
  MoveL 224 to (176.09, 221.76, 0) mm, rotated rx 180 ry 0 rz -39.83 deg; joints [49.211, -63.184, 67.713, -0.863, 85.49, 49.275]
  MoveL 225 to (176.01, 221.82, 0) mm, rotated rx 180 ry 0 rz -39.83 deg; joints [49.207, -63.179, 67.705, -0.863, 85.493, 49.272]
  MoveL 226 to (175.93, 221.88, 0) mm, rotated rx -180 ry 0 rz -39.83 deg; joints [49.203, -63.173, 67.696, -0.863, 85.495, 49.268]
  MoveL 227 to (175.86, 221.95, 0) mm, rotated rx -180 ry 0 rz -39.83 deg; joints [49.2, -63.167, 67.688, -0.863, 85.498, 49.265]
  MoveL 228 to (175.86, 221.95, 0) mm, rotated rx -180 ry 0 rz -39.83 deg; joints [49.2, -63.167, 67.688, -0.863, 85.498, 49.265]
  MoveL 229 to (177.95, 223.61, 0) mm, rotated rx 180 ry 0 rz -39.83 deg; joints [49.298, -63.022, 67.479, -0.863, 85.564, 49.362]
  MoveL 230 to (179.84, 225.48, 0) mm, rotated rx 180 ry 0 rz -39.83 deg; joints [49.388, -62.858, 67.241, -0.863, 85.639, 49.45]
  MoveL 231 to (181.53, 227.54, 0) mm, rotated rx -180 ry 0 rz -39.83 deg; joints [49.467, -62.677, 66.977, -0.863, 85.723, 49.528]
  MoveL 232 to (182.99, 229.78, 0) mm, rotated rx 180 ry 0 rz -39.83 deg; joints [49.535, -62.479, 66.688, -0.863, 85.815, 49.595]
  MoveL 233 to (182.99, 229.78, 0) mm, rotated rx 180 ry 0 rz -39.83 deg; joints [49.535, -62.479, 66.688, -0.863, 85.815, 49.595]
  MoveL 234 to (182.39, 229.77, 0) mm, rotated rx 180 ry 0 rz -39.83 deg; joints [49.508, -62.479, 66.687, -0.863, 85.815, 49.568]
  MoveL 235 to (181.8, 229.75, 0) mm, rotated rx 180 ry 0 rz -39.83 deg; joints [49.481, -62.48, 66.689, -0.863, 85.815, 49.54]
  MoveL 236 to (181.21, 229.71, 0) mm, rotated rx -180 ry 0 rz -39.83 deg; joints [49.453, -62.483, 66.692, -0.863, 85.814, 49.513]
  MoveL 237 to (180.62, 229.64, 0) mm, rotated rx 180 ry 0 rz -39.83 deg; joints [49.426, -62.489, 66.7, -0.863, 85.811, 49.486]
  MoveL 238 to (180.22, 229.57, 0) mm, rotated rx 180 ry 0 rz -39.83 deg; joints [49.407, -62.495, 66.708, -0.863, 85.809, 49.467]
  MoveL 239 to (179.81, 229.5, 0) mm, rotated rx 180 ry 0 rz -39.83 deg; joints [49.389, -62.501, 66.717, -0.863, 85.806, 49.449]
  MoveL 240 to (179.41, 229.43, 0) mm, rotated rx -180 ry 0 rz -39.83 deg; joints [49.37, -62.507, 66.725, -0.863, 85.804, 49.43]
  MoveL 241 to (179, 229.38, 0) mm, rotated rx -180 ry 0 rz -39.83 deg; joints [49.351, -62.511, 66.73, -0.863, 85.802, 49.411]
  MoveL 242 to (178.58, 229.36, 0) mm, rotated rx 180 ry 0 rz -39.83 deg; joints [49.331, -62.512, 66.731, -0.863, 85.802, 49.391]
  MoveL 243 to (178.14, 229.36, 0) mm, rotated rx -180 ry 0 rz -39.83 deg; joints [49.311, -62.511, 66.73, -0.863, 85.802, 49.371]
  MoveL 244 to (177.71, 229.38, 0) mm, rotated rx -180 ry 0 rz -39.83 deg; joints [49.291, -62.509, 66.725, -0.863, 85.804, 49.351]
  MoveL 245 to (177.28, 229.41, 0) mm, rotated rx 180 ry 0 rz -39.83 deg; joints [49.271, -62.505, 66.72, -0.863, 85.806, 49.331]
  MoveL 246 to (177.28, 229.41, 0) mm, rotated rx 180 ry 0 rz -39.83 deg; joints [49.271, -62.505, 66.72, -0.863, 85.806, 49.331]
  MoveL 247 to (177.6, 230.42, 0) mm, rotated rx 180 ry 0 rz -39.83 deg; joints [49.287, -62.416, 66.589, -0.863, 85.847, 49.346]
  MoveL 248 to (177.94, 231.41, 0) mm, rotated rx -180 ry 0 rz -39.83 deg; joints [49.304, -62.328, 66.46, -0.863, 85.889, 49.362]
  MoveL 249 to (178.33, 232.38, 0) mm, rotated rx 180 ry 0 rz -39.83 deg; joints [49.322, -62.242, 66.334, -0.863, 85.929, 49.38]
  MoveL 250 to (178.79, 233.31, 0) mm, rotated rx -180 ry 0 rz -39.83 deg; joints [49.344, -62.159, 66.212, -0.863, 85.969, 49.401]
  MoveL 251 to (179.17, 233.95, 0) mm, rotated rx 180 ry 0 rz -39.83 deg; joints [49.362, -62.102, 66.128, -0.862, 85.996, 49.419]
  MoveL 252 to (179.58, 234.58, 0) mm, rotated rx 180 ry 0 rz -39.83 deg; joints [49.381, -62.046, 66.046, -0.862, 86.022, 49.438]
  MoveL 253 to (180.02, 235.2, 0) mm, rotated rx 180 ry 0 rz -39.83 deg; joints [49.402, -61.992, 65.966, -0.862, 86.048, 49.458]
  MoveL 254 to (180.46, 235.81, 0) mm, rotated rx 180 ry 0 rz -39.83 deg; joints [49.422, -61.938, 65.886, -0.862, 86.074, 49.479]
  MoveL 255 to (180.9, 236.4, 0) mm, rotated rx 180 ry 0 rz -39.83 deg; joints [49.443, -61.885, 65.808, -0.862, 86.099, 49.498]
  MoveL 256 to (181.33, 236.99, 0) mm, rotated rx 180 ry 0 rz -39.83 deg; joints [49.463, -61.832, 65.731, -0.862, 86.124, 49.518]
  MoveL 257 to (181.76, 237.59, 0) mm, rotated rx 180 ry 0 rz -39.83 deg; joints [49.483, -61.779, 65.653, -0.862, 86.149, 49.538]
  MoveL 258 to (182.18, 238.18, 0) mm, rotated rx 180 ry 0 rz -39.83 deg; joints [49.503, -61.726, 65.575, -0.862, 86.175, 49.557]
  MoveL 259 to (182.18, 238.18, 0) mm, rotated rx 180 ry 0 rz -39.83 deg; joints [49.503, -61.726, 65.575, -0.862, 86.175, 49.557]
  MoveL 260 to (181.08, 238.2, 0) mm, rotated rx 180 ry 0 rz -39.83 deg; joints [49.452, -61.724, 65.57, -0.862, 86.176, 49.506]
  MoveL 261 to (179.97, 238.21, 0) mm, rotated rx 180 ry 0 rz -39.83 deg; joints [49.401, -61.721, 65.565, -0.862, 86.178, 49.456]
  MoveL 262 to (178.86, 238.22, 0) mm, rotated rx -180 ry 0 rz -39.83 deg; joints [49.35, -61.719, 65.56, -0.862, 86.18, 49.405]
  MoveL 263 to (177.75, 238.24, 0) mm, rotated rx 180 ry 0 rz -39.83 deg; joints [49.3, -61.716, 65.555, -0.862, 86.182, 49.354]
  MoveL 264 to (176.94, 238.25, 0) mm, rotated rx 180 ry 0 rz -39.83 deg; joints [49.262, -61.714, 65.551, -0.862, 86.183, 49.316]
  MoveL 265 to (176.12, 238.26, 0) mm, rotated rx -180 ry 0 rz -39.83 deg; joints [49.225, -61.712, 65.547, -0.862, 86.185, 49.279]
  MoveL 266 to (175.3, 238.26, 0) mm, rotated rx -180 ry 0 rz -39.83 deg; joints [49.187, -61.711, 65.544, -0.862, 86.186, 49.241]
  MoveL 267 to (174.47, 238.26, 0) mm, rotated rx 180 ry 0 rz -39.83 deg; joints [49.149, -61.71, 65.541, -0.862, 86.187, 49.203]
  MoveL 268 to (173.98, 238.26, 0) mm, rotated rx 180 ry 0 rz -39.83 deg; joints [49.126, -61.709, 65.539, -0.862, 86.188, 49.181]
  MoveL 269 to (173.48, 238.27, 0) mm, rotated rx -180 ry 0 rz -39.83 deg; joints [49.103, -61.708, 65.537, -0.862, 86.189, 49.158]
  MoveL 270 to (172.98, 238.3, 0) mm, rotated rx 180 ry 0 rz -39.83 deg; joints [49.081, -61.705, 65.531, -0.862, 86.19, 49.135]
  MoveL 271 to (172.49, 238.36, 0) mm, rotated rx 180 ry 0 rz -39.83 deg; joints [49.058, -61.698, 65.521, -0.862, 86.194, 49.112]
  MoveL 272 to (172.15, 238.42, 0) mm, rotated rx 180 ry 0 rz -39.83 deg; joints [49.043, -61.692, 65.511, -0.862, 86.197, 49.097]
  MoveL 273 to (171.8, 238.51, 0) mm, rotated rx 180 ry 0 rz -39.83 deg; joints [49.027, -61.683, 65.498, -0.862, 86.201, 49.081]
  MoveL 274 to (171.46, 238.61, 0) mm, rotated rx 180 ry 0 rz -39.83 deg; joints [49.011, -61.674, 65.484, -0.862, 86.206, 49.065]
  MoveL 275 to (171.12, 238.71, 0) mm, rotated rx -180 ry 0 rz -39.83 deg; joints [48.996, -61.664, 65.469, -0.862, 86.211, 49.05]
  MoveL 276 to (171.12, 238.71, 0) mm, rotated rx -180 ry 0 rz -39.83 deg; joints [48.996, -61.664, 65.469, -0.862, 86.211, 49.05]
  MoveL 277 to (171.43, 239.09, 0) mm, rotated rx 180 ry 0 rz -39.83 deg; joints [49.01, -61.63, 65.419, -0.862, 86.227, 49.064]
  MoveL 278 to (171.74, 239.47, 0) mm, rotated rx 180 ry 0 rz -39.83 deg; joints [49.025, -61.597, 65.37, -0.862, 86.243, 49.078]
  MoveL 279 to (172.07, 239.82, 0) mm, rotated rx -180 ry 0 rz -39.83 deg; joints [49.04, -61.566, 65.324, -0.862, 86.258, 49.094]
  MoveL 280 to (172.44, 240.15, 0) mm, rotated rx -180 ry 0 rz -39.83 deg; joints [49.058, -61.537, 65.281, -0.862, 86.272, 49.111]
  MoveL 281 to (172.78, 240.41, 0) mm, rotated rx 180 ry 0 rz -39.83 deg; joints [49.074, -61.514, 65.248, -0.862, 86.283, 49.126]
  MoveL 282 to (173.13, 240.66, 0) mm, rotated rx -180 ry 0 rz -39.83 deg; joints [49.089, -61.492, 65.215, -0.862, 86.294, 49.142]
  MoveL 283 to (173.44, 240.94, 0) mm, rotated rx -180 ry 0 rz -39.83 deg; joints [49.104, -61.467, 65.179, -0.862, 86.305, 49.157]
  MoveL 284 to (173.69, 241.26, 0) mm, rotated rx -180 ry 0 rz -39.83 deg; joints [49.116, -61.438, 65.137, -0.862, 86.319, 49.168]
  MoveL 285 to (173.75, 241.36, 0) mm, rotated rx -180 ry 0 rz -39.83 deg; joints [49.118, -61.43, 65.124, -0.862, 86.323, 49.171]
  MoveL 286 to (173.8, 241.46, 0) mm, rotated rx 180 ry 0 rz -39.83 deg; joints [49.121, -61.421, 65.111, -0.862, 86.328, 49.173]
  MoveL 287 to (173.84, 241.56, 0) mm, rotated rx 180 ry 0 rz -39.83 deg; joints [49.123, -61.412, 65.097, -0.862, 86.332, 49.175]
  MoveL 288 to (173.88, 241.66, 0) mm, rotated rx 180 ry 0 rz -39.83 deg; joints [49.125, -61.403, 65.084, -0.862, 86.337, 49.177]
  MoveL 289 to (173.88, 241.66, 0) mm, rotated rx 180 ry 0 rz -39.83 deg; joints [49.125, -61.403, 65.084, -0.862, 86.337, 49.177]
  MoveL 290 to (173.25, 241.73, 0) mm, rotated rx 180 ry 0 rz -39.83 deg; joints [49.096, -61.396, 65.072, -0.862, 86.34, 49.148]
  MoveL 291 to (172.61, 241.79, 0) mm, rotated rx -180 ry 0 rz -39.83 deg; joints [49.067, -61.389, 65.062, -0.862, 86.344, 49.119]
  MoveL 292 to (171.97, 241.85, 0) mm, rotated rx 180 ry 0 rz -39.83 deg; joints [49.037, -61.383, 65.052, -0.862, 86.347, 49.089]
  MoveL 293 to (171.33, 241.9, 0) mm, rotated rx 180 ry 0 rz -39.83 deg; joints [49.008, -61.377, 65.043, -0.862, 86.35, 49.06]
  MoveL 294 to (170.26, 241.95, 0) mm, rotated rx 180 ry 0 rz -39.83 deg; joints [48.96, -61.371, 65.031, -0.862, 86.354, 49.011]
  MoveL 295 to (169.19, 241.97, 0) mm, rotated rx 180 ry 0 rz -39.83 deg; joints [48.911, -61.367, 65.025, -0.862, 86.357, 48.962]
  MoveL 296 to (168.12, 241.95, 0) mm, rotated rx 180 ry 0 rz -39.83 deg; joints [48.862, -61.367, 65.024, -0.862, 86.357, 48.913]
  MoveL 297 to (167.05, 241.88, 0) mm, rotated rx 180 ry 0 rz -39.83 deg; joints [48.813, -61.371, 65.029, -0.862, 86.356, 48.864]
  MoveL 298 to (166.28, 241.79, 0) mm, rotated rx 180 ry 0 rz -39.83 deg; joints [48.777, -61.377, 65.036, -0.862, 86.353, 48.829]
  MoveL 299 to (165.51, 241.67, 0) mm, rotated rx -180 ry 0 rz -39.83 deg; joints [48.742, -61.387, 65.049, -0.862, 86.349, 48.793]
  MoveL 300 to (164.75, 241.49, 0) mm, rotated rx 180 ry 0 rz -39.83 deg; joints [48.707, -61.401, 65.07, -0.862, 86.343, 48.759]
  MoveL 301 to (164.02, 241.24, 0) mm, rotated rx -180 ry 0 rz -39.83 deg; joints [48.673, -61.423, 65.101, -0.862, 86.333, 48.725]
  MoveL 302 to (163.51, 241, 0) mm, rotated rx 180 ry 0 rz -39.83 deg; joints [48.649, -61.443, 65.13, -0.862, 86.323, 48.702]
  MoveL 303 to (163, 240.75, 0) mm, rotated rx -180 ry 0 rz -39.83 deg; joints [48.626, -61.465, 65.162, -0.862, 86.313, 48.678]
  MoveL 304 to (162.48, 240.5, 0) mm, rotated rx 180 ry 0 rz -39.83 deg; joints [48.602, -61.486, 65.193, -0.862, 86.303, 48.654]
  MoveL 305 to (161.96, 240.29, 0) mm, rotated rx 180 ry 0 rz -39.83 deg; joints [48.578, -61.504, 65.218, -0.862, 86.295, 48.63]
  MoveL 306 to (161.7, 240.21, 0) mm, rotated rx 180 ry 0 rz -39.83 deg; joints [48.566, -61.51, 65.228, -0.862, 86.291, 48.619]
  MoveL 307 to (161.45, 240.14, 0) mm, rotated rx 180 ry 0 rz -39.83 deg; joints [48.554, -61.516, 65.236, -0.862, 86.289, 48.607]
  MoveL 308 to (161.19, 240.08, 0) mm, rotated rx 180 ry 0 rz -39.83 deg; joints [48.542, -61.521, 65.243, -0.862, 86.287, 48.595]
  MoveL 309 to (160.93, 240.02, 0) mm, rotated rx -180 ry 0 rz -39.83 deg; joints [48.53, -61.525, 65.249, -0.862, 86.285, 48.583]
  MoveL 310 to (160.93, 240.02, 0) mm, rotated rx -180 ry 0 rz -39.83 deg; joints [48.53, -61.525, 65.249, -0.862, 86.285, 48.583]
  MoveL 311 to (160.8, 240.36, 0) mm, rotated rx 180 ry 0 rz -39.83 deg; joints [48.525, -61.494, 65.203, -0.862, 86.3, 48.577]
  MoveL 312 to (160.7, 240.7, 0) mm, rotated rx -180 ry 0 rz -39.83 deg; joints [48.52, -61.463, 65.157, -0.862, 86.315, 48.573]
  MoveL 313 to (160.64, 241.04, 0) mm, rotated rx 180 ry 0 rz -39.83 deg; joints [48.518, -61.433, 65.111, -0.862, 86.33, 48.57]
  MoveL 314 to (160.65, 241.37, 0) mm, rotated rx 180 ry 0 rz -39.83 deg; joints [48.519, -61.403, 65.068, -0.862, 86.344, 48.571]
  MoveL 315 to (160.75, 241.7, 0) mm, rotated rx 180 ry 0 rz -39.83 deg; joints [48.524, -61.373, 65.023, -0.862, 86.359, 48.576]
  MoveL 316 to (160.94, 242.02, 0) mm, rotated rx 180 ry 0 rz -39.83 deg; joints [48.533, -61.345, 64.982, -0.862, 86.372, 48.585]
  MoveL 317 to (161.18, 242.31, 0) mm, rotated rx 180 ry 0 rz -39.83 deg; joints [48.545, -61.32, 64.944, -0.862, 86.385, 48.596]
  MoveL 318 to (161.46, 242.58, 0) mm, rotated rx 180 ry 0 rz -39.83 deg; joints [48.558, -61.296, 64.909, -0.862, 86.396, 48.609]
  MoveL 319 to (161.68, 242.76, 0) mm, rotated rx -180 ry 0 rz -39.83 deg; joints [48.568, -61.28, 64.885, -0.862, 86.404, 48.619]
  MoveL 320 to (161.9, 242.94, 0) mm, rotated rx 180 ry 0 rz -39.83 deg; joints [48.578, -61.264, 64.863, -0.862, 86.411, 48.629]
  MoveL 321 to (162.13, 243.1, 0) mm, rotated rx 180 ry 0 rz -39.83 deg; joints [48.589, -61.25, 64.841, -0.862, 86.418, 48.64]
  MoveL 322 to (162.36, 243.26, 0) mm, rotated rx -180 ry 0 rz -39.83 deg; joints [48.6, -61.236, 64.821, -0.862, 86.425, 48.65]
  MoveL 323 to (162.61, 243.44, 0) mm, rotated rx 180 ry 0 rz -39.83 deg; joints [48.611, -61.221, 64.799, -0.862, 86.432, 48.662]
  MoveL 324 to (162.86, 243.61, 0) mm, rotated rx -180 ry 0 rz -39.83 deg; joints [48.623, -61.206, 64.776, -0.862, 86.44, 48.673]
  MoveL 325 to (163.11, 243.79, 0) mm, rotated rx 180 ry 0 rz -39.83 deg; joints [48.635, -61.19, 64.753, -0.862, 86.447, 48.685]
  MoveL 326 to (163.35, 243.98, 0) mm, rotated rx -180 ry 0 rz -39.83 deg; joints [48.646, -61.174, 64.73, -0.862, 86.455, 48.696]
  MoveL 327 to (163.48, 244.07, 0) mm, rotated rx -180 ry 0 rz -39.83 deg; joints [48.652, -61.166, 64.718, -0.862, 86.459, 48.702]
  MoveL 328 to (163.6, 244.16, 0) mm, rotated rx -180 ry 0 rz -39.83 deg; joints [48.658, -61.158, 64.705, -0.862, 86.463, 48.708]
  MoveL 329 to (163.73, 244.26, 0) mm, rotated rx 180 ry 0 rz -39.83 deg; joints [48.663, -61.149, 64.693, -0.862, 86.467, 48.713]
  MoveL 330 to (163.85, 244.35, 0) mm, rotated rx 180 ry 0 rz -39.83 deg; joints [48.669, -61.141, 64.681, -0.862, 86.471, 48.719]
  MoveL 331 to (163.85, 244.35, 0) mm, rotated rx 180 ry 0 rz -39.83 deg; joints [48.669, -61.141, 64.681, -0.862, 86.471, 48.719]
  MoveL 332 to (163.12, 244.34, 0) mm, rotated rx 180 ry 0 rz -39.83 deg; joints [48.636, -61.14, 64.679, -0.862, 86.471, 48.686]
  MoveL 333 to (162.38, 244.31, 0) mm, rotated rx -180 ry 0 rz -39.83 deg; joints [48.602, -61.141, 64.68, -0.862, 86.471, 48.652]
  MoveL 334 to (161.65, 244.25, 0) mm, rotated rx 180 ry 0 rz -39.83 deg; joints [48.569, -61.145, 64.684, -0.862, 86.47, 48.619]
  MoveL 335 to (160.93, 244.15, 0) mm, rotated rx 180 ry 0 rz -39.83 deg; joints [48.536, -61.153, 64.694, -0.862, 86.467, 48.586]
  MoveL 336 to (160.38, 244.04, 0) mm, rotated rx 180 ry 0 rz -39.83 deg; joints [48.511, -61.162, 64.707, -0.862, 86.463, 48.561]
  MoveL 337 to (159.84, 243.9, 0) mm, rotated rx 180 ry 0 rz -39.83 deg; joints [48.485, -61.172, 64.723, -0.862, 86.458, 48.536]
  MoveL 338 to (159.29, 243.76, 0) mm, rotated rx -180 ry 0 rz -39.83 deg; joints [48.46, -61.184, 64.739, -0.862, 86.453, 48.511]
  MoveL 339 to (158.75, 243.63, 0) mm, rotated rx 180 ry 0 rz -39.83 deg; joints [48.435, -61.194, 64.754, -0.862, 86.448, 48.485]
  MoveL 340 to (158.4, 243.56, 0) mm, rotated rx -180 ry 0 rz -39.83 deg; joints [48.419, -61.2, 64.762, -0.862, 86.445, 48.469]
  MoveL 341 to (158.05, 243.49, 0) mm, rotated rx 180 ry 0 rz -39.83 deg; joints [48.403, -61.205, 64.769, -0.862, 86.443, 48.453]
  MoveL 342 to (157.7, 243.41, 0) mm, rotated rx 180 ry 0 rz -39.83 deg; joints [48.387, -61.211, 64.777, -0.862, 86.44, 48.437]
  MoveL 343 to (157.35, 243.33, 0) mm, rotated rx 180 ry 0 rz -39.83 deg; joints [48.371, -61.217, 64.786, -0.862, 86.437, 48.421]
  MoveL 344 to (156.88, 243.2, 0) mm, rotated rx 180 ry 0 rz -39.83 deg; joints [48.349, -61.228, 64.802, -0.862, 86.432, 48.4]
  MoveL 345 to (156.41, 243.05, 0) mm, rotated rx -180 ry 0 rz -39.83 deg; joints [48.328, -61.24, 64.82, -0.862, 86.426, 48.378]
  MoveL 346 to (155.95, 242.89, 0) mm, rotated rx 180 ry 0 rz -39.83 deg; joints [48.307, -61.254, 64.839, -0.862, 86.42, 48.357]
  MoveL 347 to (155.49, 242.72, 0) mm, rotated rx 180 ry 0 rz -39.83 deg; joints [48.285, -61.267, 64.858, -0.862, 86.414, 48.336]
  MoveL 348 to (155.07, 242.58, 0) mm, rotated rx 180 ry 0 rz -39.83 deg; joints [48.266, -61.279, 64.875, -0.862, 86.408, 48.317]
  MoveL 349 to (154.65, 242.44, 0) mm, rotated rx 180 ry 0 rz -39.83 deg; joints [48.246, -61.29, 64.891, -0.862, 86.403, 48.297]
  MoveL 350 to (154.22, 242.31, 0) mm, rotated rx 180 ry 0 rz -39.83 deg; joints [48.227, -61.301, 64.907, -0.862, 86.398, 48.278]
  MoveL 351 to (153.8, 242.19, 0) mm, rotated rx 180 ry 0 rz -39.83 deg; joints [48.207, -61.311, 64.921, -0.862, 86.394, 48.258]
  MoveL 352 to (153.56, 242.13, 0) mm, rotated rx 180 ry 0 rz -39.83 deg; joints [48.196, -61.316, 64.928, -0.862, 86.391, 48.247]
  MoveL 353 to (153.33, 242.07, 0) mm, rotated rx 180 ry 0 rz -39.83 deg; joints [48.185, -61.32, 64.935, -0.862, 86.389, 48.237]
  MoveL 354 to (153.09, 242.01, 0) mm, rotated rx 180 ry 0 rz -39.83 deg; joints [48.175, -61.324, 64.941, -0.862, 86.387, 48.226]
  MoveL 355 to (152.86, 241.97, 0) mm, rotated rx -180 ry 0 rz -39.83 deg; joints [48.164, -61.328, 64.945, -0.862, 86.386, 48.215]
  MoveL 356 to (152.7, 241.94, 0) mm, rotated rx 180 ry 0 rz -39.83 deg; joints [48.156, -61.33, 64.948, -0.862, 86.385, 48.207]
  MoveL 357 to (152.53, 241.92, 0) mm, rotated rx -180 ry 0 rz -39.83 deg; joints [48.149, -61.331, 64.95, -0.862, 86.384, 48.2]
  MoveL 358 to (152.37, 241.9, 0) mm, rotated rx 180 ry 0 rz -39.83 deg; joints [48.141, -61.333, 64.952, -0.862, 86.384, 48.192]
  MoveL 359 to (152.2, 241.88, 0) mm, rotated rx 180 ry 0 rz -39.83 deg; joints [48.134, -61.334, 64.954, -0.862, 86.383, 48.185]
  MoveL 360 to (152.2, 241.88, 0) mm, rotated rx 180 ry 0 rz -39.83 deg; joints [48.134, -61.334, 64.954, -0.862, 86.383, 48.185]
  MoveL 361 to (152.2, 242.16, 0) mm, rotated rx 180 ry 0 rz -39.83 deg; joints [48.134, -61.309, 64.916, -0.862, 86.395, 48.185]
  MoveL 362 to (152.21, 242.43, 0) mm, rotated rx 180 ry 0 rz -39.83 deg; joints [48.135, -61.284, 64.879, -0.862, 86.408, 48.186]
  MoveL 363 to (152.24, 242.7, 0) mm, rotated rx 180 ry 0 rz -39.83 deg; joints [48.137, -61.26, 64.843, -0.862, 86.419, 48.188]
  MoveL 364 to (152.31, 242.96, 0) mm, rotated rx 180 ry 0 rz -39.83 deg; joints [48.14, -61.236, 64.808, -0.862, 86.431, 48.191]
  MoveL 365 to (152.41, 243.2, 0) mm, rotated rx -180 ry 0 rz -39.83 deg; joints [48.145, -61.215, 64.776, -0.862, 86.441, 48.196]
  MoveL 366 to (152.54, 243.43, 0) mm, rotated rx -180 ry 0 rz -39.83 deg; joints [48.152, -61.195, 64.746, -0.862, 86.451, 48.202]
  MoveL 367 to (152.7, 243.65, 0) mm, rotated rx 180 ry 0 rz -39.83 deg; joints [48.159, -61.175, 64.718, -0.862, 86.461, 48.209]
  MoveL 368 to (152.87, 243.85, 0) mm, rotated rx -180 ry 0 rz -39.83 deg; joints [48.167, -61.157, 64.691, -0.862, 86.469, 48.217]
  MoveL 369 to (153.18, 244.16, 0) mm, rotated rx 180 ry 0 rz -39.83 deg; joints [48.182, -61.131, 64.652, -0.862, 86.482, 48.232]
  MoveL 370 to (153.51, 244.44, 0) mm, rotated rx 180 ry 0 rz -39.83 deg; joints [48.198, -61.106, 64.616, -0.862, 86.494, 48.247]
  MoveL 371 to (153.86, 244.7, 0) mm, rotated rx 180 ry 0 rz -39.83 deg; joints [48.214, -61.084, 64.582, -0.862, 86.505, 48.263]
  MoveL 372 to (154.21, 244.95, 0) mm, rotated rx 180 ry 0 rz -39.83 deg; joints [48.23, -61.062, 64.551, -0.862, 86.516, 48.279]
  MoveL 373 to (154.42, 245.1, 0) mm, rotated rx 180 ry 0 rz -39.83 deg; joints [48.24, -61.049, 64.532, -0.862, 86.522, 48.289]
  MoveL 374 to (154.63, 245.24, 0) mm, rotated rx 180 ry 0 rz -39.83 deg; joints [48.25, -61.037, 64.514, -0.862, 86.528, 48.299]
  MoveL 375 to (154.85, 245.39, 0) mm, rotated rx 180 ry 0 rz -39.83 deg; joints [48.26, -61.024, 64.495, -0.862, 86.534, 48.309]
  MoveL 376 to (155.06, 245.53, 0) mm, rotated rx -180 ry 0 rz -39.83 deg; joints [48.27, -61.012, 64.477, -0.862, 86.54, 48.319]
  MoveL 377 to (155.27, 245.67, 0) mm, rotated rx -180 ry 0 rz -39.83 deg; joints [48.28, -61, 64.459, -0.862, 86.546, 48.328]
  MoveL 378 to (155.48, 245.81, 0) mm, rotated rx 180 ry 0 rz -39.83 deg; joints [48.289, -60.988, 64.441, -0.862, 86.552, 48.338]
  MoveL 379 to (155.69, 245.96, 0) mm, rotated rx 180 ry 0 rz -39.83 deg; joints [48.299, -60.975, 64.423, -0.862, 86.557, 48.348]
  MoveL 380 to (155.91, 246.1, 0) mm, rotated rx -180 ry 0 rz -39.83 deg; joints [48.309, -60.963, 64.405, -0.862, 86.563, 48.358]
  MoveL 381 to (155.91, 246.1, 0) mm, rotated rx -180 ry 0 rz -39.83 deg; joints [48.309, -60.963, 64.405, -0.862, 86.563, 48.358]
  MoveL 382 to (155, 246.07, 0) mm, rotated rx 180 ry 0 rz -39.83 deg; joints [48.268, -60.963, 64.403, -0.862, 86.564, 48.317]
  MoveL 383 to (154.1, 246.03, 0) mm, rotated rx 180 ry 0 rz -39.83 deg; joints [48.227, -60.964, 64.404, -0.862, 86.564, 48.275]
  MoveL 384 to (153.21, 245.95, 0) mm, rotated rx 180 ry 0 rz -39.83 deg; joints [48.186, -60.969, 64.41, -0.862, 86.562, 48.235]
  MoveL 385 to (152.33, 245.81, 0) mm, rotated rx 180 ry 0 rz -39.83 deg; joints [48.146, -60.979, 64.424, -0.862, 86.558, 48.194]
  MoveL 386 to (151.54, 245.62, 0) mm, rotated rx -180 ry 0 rz -39.83 deg; joints [48.11, -60.994, 64.445, -0.862, 86.551, 48.158]
  MoveL 387 to (150.76, 245.37, 0) mm, rotated rx 180 ry 0 rz -39.83 deg; joints [48.074, -61.013, 64.474, -0.862, 86.542, 48.123]
  MoveL 388 to (150, 245.09, 0) mm, rotated rx 180 ry 0 rz -39.83 deg; joints [48.038, -61.037, 64.507, -0.862, 86.531, 48.087]
  MoveL 389 to (149.24, 244.78, 0) mm, rotated rx -180 ry 0 rz -39.83 deg; joints [48.003, -61.062, 64.545, -0.862, 86.518, 48.052]
  MoveL 390 to (148.74, 244.57, 0) mm, rotated rx 180 ry 0 rz -39.83 deg; joints [47.98, -61.08, 64.57, -0.862, 86.51, 48.03]
  MoveL 391 to (148.25, 244.34, 0) mm, rotated rx 180 ry 0 rz -39.83 deg; joints [47.957, -61.098, 64.597, -0.862, 86.501, 48.007]
  MoveL 392 to (147.77, 244.11, 0) mm, rotated rx 180 ry 0 rz -39.83 deg; joints [47.935, -61.118, 64.626, -0.862, 86.492, 47.985]
  MoveL 393 to (147.29, 243.86, 0) mm, rotated rx -180 ry 0 rz -39.83 deg; joints [47.913, -61.139, 64.656, -0.862, 86.482, 47.963]
  MoveL 394 to (146.84, 243.61, 0) mm, rotated rx 180 ry 0 rz -39.83 deg; joints [47.892, -61.16, 64.687, -0.862, 86.472, 47.941]
  MoveL 395 to (146.39, 243.34, 0) mm, rotated rx 180 ry 0 rz -39.83 deg; joints [47.871, -61.182, 64.72, -0.862, 86.461, 47.921]
  MoveL 396 to (145.94, 243.07, 0) mm, rotated rx -180 ry 0 rz -39.83 deg; joints [47.85, -61.206, 64.754, -0.862, 86.45, 47.9]
  MoveL 397 to (145.5, 242.8, 0) mm, rotated rx 180 ry 0 rz -39.83 deg; joints [47.829, -61.229, 64.788, -0.862, 86.439, 47.879]
  MoveL 398 to (145.2, 242.61, 0) mm, rotated rx 180 ry 0 rz -39.83 deg; joints [47.815, -61.244, 64.811, -0.862, 86.431, 47.866]
  MoveL 399 to (144.91, 242.43, 0) mm, rotated rx 180 ry 0 rz -39.83 deg; joints [47.801, -61.259, 64.833, -0.862, 86.424, 47.852]
  MoveL 400 to (144.61, 242.25, 0) mm, rotated rx -180 ry 0 rz -39.83 deg; joints [47.788, -61.275, 64.856, -0.862, 86.417, 47.838]
  MoveL 401 to (144.32, 242.07, 0) mm, rotated rx -180 ry 0 rz -39.83 deg; joints [47.774, -61.29, 64.878, -0.862, 86.409, 47.824]
  MoveL 402 to (144.32, 242.07, 0) mm, rotated rx -180 ry 0 rz -39.83 deg; joints [47.774, -61.29, 64.878, -0.862, 86.409, 47.824]
  MoveL 403 to (144.13, 242.41, 0) mm, rotated rx 180 ry 0 rz -39.83 deg; joints [47.766, -61.259, 64.831, -0.862, 86.425, 47.816]
  MoveL 404 to (143.97, 242.75, 0) mm, rotated rx 180 ry 0 rz -39.83 deg; joints [47.759, -61.227, 64.784, -0.862, 86.44, 47.81]
  MoveL 405 to (143.86, 243.1, 0) mm, rotated rx -180 ry 0 rz -39.83 deg; joints [47.755, -61.196, 64.737, -0.862, 86.456, 47.805]
  MoveL 406 to (143.81, 243.45, 0) mm, rotated rx 180 ry 0 rz -39.83 deg; joints [47.753, -61.164, 64.689, -0.862, 86.472, 47.803]
  MoveL 407 to (143.85, 243.78, 0) mm, rotated rx 180 ry 0 rz -39.83 deg; joints [47.756, -61.134, 64.645, -0.862, 86.486, 47.805]
  MoveL 408 to (143.95, 244.11, 0) mm, rotated rx -180 ry 0 rz -39.83 deg; joints [47.761, -61.105, 64.601, -0.862, 86.501, 47.81]
  MoveL 409 to (144.1, 244.43, 0) mm, rotated rx 180 ry 0 rz -39.83 deg; joints [47.768, -61.076, 64.559, -0.862, 86.515, 47.817]
  MoveL 410 to (144.28, 244.73, 0) mm, rotated rx 180 ry 0 rz -39.83 deg; joints [47.777, -61.05, 64.519, -0.862, 86.528, 47.826]
  MoveL 411 to (144.46, 244.98, 0) mm, rotated rx 180 ry 0 rz -39.83 deg; joints [47.786, -61.027, 64.486, -0.862, 86.539, 47.835]
  MoveL 412 to (144.65, 245.23, 0) mm, rotated rx 180 ry 0 rz -39.83 deg; joints [47.795, -61.006, 64.455, -0.862, 86.549, 47.844]
  MoveL 413 to (144.85, 245.46, 0) mm, rotated rx 180 ry 0 rz -39.83 deg; joints [47.804, -60.986, 64.425, -0.862, 86.559, 47.853]
  MoveL 414 to (145.05, 245.69, 0) mm, rotated rx 180 ry 0 rz -39.83 deg; joints [47.814, -60.966, 64.395, -0.862, 86.569, 47.863]
  MoveL 415 to (145.25, 245.91, 0) mm, rotated rx -180 ry 0 rz -39.83 deg; joints [47.824, -60.946, 64.366, -0.862, 86.578, 47.872]
  MoveL 416 to (145.45, 246.13, 0) mm, rotated rx 180 ry 0 rz -39.83 deg; joints [47.833, -60.927, 64.337, -0.862, 86.588, 47.881]
  MoveL 417 to (145.65, 246.36, 0) mm, rotated rx 180 ry 0 rz -39.83 deg; joints [47.842, -60.907, 64.308, -0.862, 86.597, 47.89]
  MoveL 418 to (145.85, 246.58, 0) mm, rotated rx -180 ry 0 rz -39.83 deg; joints [47.852, -60.887, 64.279, -0.862, 86.607, 47.9]
  MoveL 419 to (145.85, 246.58, 0) mm, rotated rx -180 ry 0 rz -39.83 deg; joints [47.852, -60.887, 64.279, -0.862, 86.607, 47.9]
  MoveL 420 to (145.43, 246.54, 0) mm, rotated rx 180 ry 0 rz -39.83 deg; joints [47.833, -60.889, 64.281, -0.862, 86.606, 47.881]
  MoveL 421 to (145.02, 246.5, 0) mm, rotated rx 180 ry 0 rz -39.83 deg; joints [47.814, -60.892, 64.285, -0.862, 86.605, 47.862]
  MoveL 422 to (144.62, 246.43, 0) mm, rotated rx 180 ry 0 rz -39.83 deg; joints [47.796, -60.896, 64.291, -0.862, 86.603, 47.844]
  MoveL 423 to (144.22, 246.34, 0) mm, rotated rx 180 ry 0 rz -39.83 deg; joints [47.777, -60.903, 64.3, -0.862, 86.6, 47.825]
  MoveL 424 to (143.69, 246.18, 0) mm, rotated rx 180 ry 0 rz -39.83 deg; joints [47.753, -60.916, 64.319, -0.862, 86.594, 47.801]
  MoveL 425 to (143.18, 245.97, 0) mm, rotated rx 180 ry 0 rz -39.83 deg; joints [47.729, -60.933, 64.344, -0.862, 86.586, 47.777]
  MoveL 426 to (142.68, 245.73, 0) mm, rotated rx -180 ry 0 rz -39.83 deg; joints [47.706, -60.953, 64.373, -0.862, 86.576, 47.754]
  MoveL 427 to (142.19, 245.46, 0) mm, rotated rx 180 ry 0 rz -39.83 deg; joints [47.683, -60.975, 64.406, -0.862, 86.566, 47.731]
  MoveL 428 to (141.93, 245.32, 0) mm, rotated rx 180 ry 0 rz -39.83 deg; joints [47.671, -60.987, 64.423, -0.862, 86.56, 47.72]
  MoveL 429 to (141.69, 245.18, 0) mm, rotated rx 180 ry 0 rz -39.83 deg; joints [47.66, -60.999, 64.441, -0.862, 86.554, 47.708]
  MoveL 430 to (141.44, 245.03, 0) mm, rotated rx -180 ry 0 rz -39.83 deg; joints [47.648, -61.012, 64.459, -0.862, 86.548, 47.697]
  MoveL 431 to (141.2, 244.87, 0) mm, rotated rx -180 ry 0 rz -39.83 deg; joints [47.637, -61.025, 64.478, -0.862, 86.542, 47.686]
  MoveL 432 to (140.84, 244.62, 0) mm, rotated rx 180 ry 0 rz -39.83 deg; joints [47.62, -61.047, 64.51, -0.862, 86.531, 47.669]
  MoveL 433 to (140.49, 244.35, 0) mm, rotated rx 180 ry 0 rz -39.83 deg; joints [47.604, -61.07, 64.544, -0.862, 86.52, 47.653]
  MoveL 434 to (140.14, 244.07, 0) mm, rotated rx 180 ry 0 rz -39.83 deg; joints [47.587, -61.093, 64.579, -0.862, 86.509, 47.636]
  MoveL 435 to (139.79, 243.8, 0) mm, rotated rx 180 ry 0 rz -39.83 deg; joints [47.571, -61.117, 64.614, -0.862, 86.497, 47.62]
  MoveL 436 to (139.43, 243.52, 0) mm, rotated rx 180 ry 0 rz -39.83 deg; joints [47.553, -61.14, 64.649, -0.862, 86.486, 47.603]
  MoveL 437 to (139.06, 243.24, 0) mm, rotated rx 180 ry 0 rz -39.83 deg; joints [47.536, -61.164, 64.683, -0.862, 86.474, 47.586]
  MoveL 438 to (138.69, 242.96, 0) mm, rotated rx 180 ry 0 rz -39.83 deg; joints [47.519, -61.188, 64.718, -0.862, 86.463, 47.569]
  MoveL 439 to (138.33, 242.68, 0) mm, rotated rx 180 ry 0 rz -39.83 deg; joints [47.502, -61.212, 64.754, -0.862, 86.451, 47.552]
  MoveL 440 to (138.03, 242.42, 0) mm, rotated rx 180 ry 0 rz -39.83 deg; joints [47.487, -61.234, 64.787, -0.862, 86.44, 47.537]
  MoveL 441 to (137.72, 242.15, 0) mm, rotated rx 180 ry 0 rz -39.83 deg; joints [47.473, -61.257, 64.82, -0.862, 86.43, 47.523]
  MoveL 442 to (137.42, 241.89, 0) mm, rotated rx 180 ry 0 rz -39.83 deg; joints [47.458, -61.28, 64.854, -0.862, 86.419, 47.509]
  MoveL 443 to (137.12, 241.63, 0) mm, rotated rx 180 ry 0 rz -39.83 deg; joints [47.444, -61.302, 64.887, -0.862, 86.408, 47.495]
  MoveL 444 to (136.88, 241.43, 0) mm, rotated rx -180 ry 0 rz -39.83 deg; joints [47.433, -61.319, 64.911, -0.862, 86.4, 47.484]
  MoveL 445 to (136.64, 241.24, 0) mm, rotated rx -180 ry 0 rz -39.83 deg; joints [47.421, -61.335, 64.935, -0.862, 86.392, 47.472]
  MoveL 446 to (136.4, 241.05, 0) mm, rotated rx 180 ry 0 rz -39.83 deg; joints [47.41, -61.351, 64.959, -0.862, 86.384, 47.461]
  MoveL 447 to (136.16, 240.86, 0) mm, rotated rx 180 ry 0 rz -39.83 deg; joints [47.399, -61.367, 64.982, -0.862, 86.377, 47.45]
  MoveL 448 to (136.16, 240.86, 0) mm, rotated rx 180 ry 0 rz -39.83 deg; joints [47.399, -61.367, 64.982, -0.862, 86.377, 47.45]
  MoveL 449 to (135.98, 241.19, 0) mm, rotated rx 180 ry 0 rz -39.83 deg; joints [47.391, -61.337, 64.937, -0.862, 86.391, 47.442]
  MoveL 450 to (135.8, 241.52, 0) mm, rotated rx 180 ry 0 rz -39.83 deg; joints [47.384, -61.307, 64.892, -0.862, 86.406, 47.435]
  MoveL 451 to (135.65, 241.85, 0) mm, rotated rx 180 ry 0 rz -39.83 deg; joints [47.378, -61.276, 64.845, -0.862, 86.422, 47.428]
  MoveL 452 to (135.54, 242.2, 0) mm, rotated rx 180 ry 0 rz -39.83 deg; joints [47.373, -61.244, 64.798, -0.862, 86.437, 47.423]
  MoveL 453 to (135.46, 242.64, 0) mm, rotated rx -180 ry 0 rz -39.83 deg; joints [47.37, -61.204, 64.738, -0.862, 86.457, 47.42]
  MoveL 454 to (135.43, 243.08, 0) mm, rotated rx 180 ry 0 rz -39.83 deg; joints [47.37, -61.164, 64.678, -0.862, 86.477, 47.42]
  MoveL 455 to (135.47, 243.53, 0) mm, rotated rx 180 ry 0 rz -39.83 deg; joints [47.373, -61.123, 64.618, -0.862, 86.497, 47.422]
  MoveL 456 to (135.56, 243.97, 0) mm, rotated rx 180 ry 0 rz -39.83 deg; joints [47.378, -61.084, 64.56, -0.862, 86.516, 47.427]
  MoveL 457 to (135.69, 244.35, 0) mm, rotated rx 180 ry 0 rz -39.83 deg; joints [47.385, -61.05, 64.508, -0.862, 86.533, 47.434]
  MoveL 458 to (135.85, 244.73, 0) mm, rotated rx 180 ry 0 rz -39.83 deg; joints [47.393, -61.017, 64.459, -0.862, 86.549, 47.442]
  MoveL 459 to (136.04, 245.09, 0) mm, rotated rx -180 ry 0 rz -39.83 deg; joints [47.402, -60.985, 64.412, -0.862, 86.565, 47.451]
  MoveL 460 to (136.23, 245.45, 0) mm, rotated rx 180 ry 0 rz -39.83 deg; joints [47.412, -60.953, 64.364, -0.862, 86.58, 47.46]
  MoveL 461 to (136.23, 245.45, 0) mm, rotated rx 180 ry 0 rz -39.83 deg; joints [47.412, -60.953, 64.364, -0.862, 86.58, 47.46]
  MoveL 462 to (135.82, 245.3, 0) mm, rotated rx -180 ry 0 rz -39.83 deg; joints [47.393, -60.965, 64.381, -0.862, 86.575, 47.441]
  MoveL 463 to (135.4, 245.14, 0) mm, rotated rx 180 ry 0 rz -39.83 deg; joints [47.373, -60.977, 64.399, -0.862, 86.569, 47.422]
  MoveL 464 to (134.99, 244.98, 0) mm, rotated rx 180 ry 0 rz -39.83 deg; joints [47.354, -60.99, 64.418, -0.862, 86.563, 47.403]
  MoveL 465 to (134.59, 244.8, 0) mm, rotated rx 180 ry 0 rz -39.83 deg; joints [47.336, -61.005, 64.44, -0.862, 86.556, 47.384]
  MoveL 466 to (134.14, 244.56, 0) mm, rotated rx 180 ry 0 rz -39.83 deg; joints [47.315, -61.024, 64.468, -0.862, 86.546, 47.363]
  MoveL 467 to (133.7, 244.3, 0) mm, rotated rx 180 ry 0 rz -39.83 deg; joints [47.294, -61.046, 64.5, -0.862, 86.536, 47.343]
  MoveL 468 to (133.27, 244.01, 0) mm, rotated rx 180 ry 0 rz -39.83 deg; joints [47.274, -61.07, 64.536, -0.862, 86.524, 47.323]
  MoveL 469 to (132.87, 243.7, 0) mm, rotated rx -180 ry 0 rz -39.83 deg; joints [47.255, -61.097, 64.575, -0.862, 86.511, 47.304]
  MoveL 470 to (132.51, 243.38, 0) mm, rotated rx 180 ry 0 rz -39.83 deg; joints [47.238, -61.124, 64.615, -0.862, 86.498, 47.287]
  MoveL 471 to (132.17, 243.05, 0) mm, rotated rx -180 ry 0 rz -39.83 deg; joints [47.221, -61.152, 64.657, -0.862, 86.484, 47.271]
  MoveL 472 to (131.83, 242.71, 0) mm, rotated rx 180 ry 0 rz -39.83 deg; joints [47.205, -61.182, 64.7, -0.862, 86.47, 47.255]
  MoveL 473 to (131.5, 242.36, 0) mm, rotated rx -180 ry 0 rz -39.83 deg; joints [47.189, -61.212, 64.745, -0.862, 86.456, 47.239]
  MoveL 474 to (131.18, 242.01, 0) mm, rotated rx 180 ry 0 rz -39.83 deg; joints [47.174, -61.242, 64.789, -0.862, 86.441, 47.224]
  MoveL 475 to (130.85, 241.66, 0) mm, rotated rx 180 ry 0 rz -39.83 deg; joints [47.158, -61.271, 64.833, -0.862, 86.427, 47.208]
  MoveL 476 to (130.53, 241.32, 0) mm, rotated rx 180 ry 0 rz -39.83 deg; joints [47.142, -61.301, 64.877, -0.862, 86.412, 47.193]
  MoveL 477 to (130.21, 240.97, 0) mm, rotated rx 180 ry 0 rz -39.83 deg; joints [47.127, -61.331, 64.921, -0.862, 86.398, 47.178]
  MoveL 478 to (130.21, 240.97, 0) mm, rotated rx 180 ry 0 rz -39.83 deg; joints [47.127, -61.331, 64.921, -0.862, 86.398, 47.178]
  MoveL 479 to (130.07, 240.8, 0) mm, rotated rx 180 ry 0 rz -39.83 deg; joints [47.12, -61.346, 64.943, -0.862, 86.391, 47.171]
  MoveL 480 to (129.93, 240.63, 0) mm, rotated rx 180 ry 0 rz -39.83 deg; joints [47.113, -61.361, 64.965, -0.862, 86.383, 47.164]
  MoveL 481 to (129.79, 240.45, 0) mm, rotated rx 180 ry 0 rz -39.83 deg; joints [47.107, -61.376, 64.987, -0.862, 86.376, 47.158]
  MoveL 482 to (129.65, 240.28, 0) mm, rotated rx 180 ry 0 rz -39.83 deg; joints [47.1, -61.391, 65.009, -0.862, 86.369, 47.151]
  MoveL 483 to (129.38, 239.93, 0) mm, rotated rx -180 ry 0 rz -39.83 deg; joints [47.087, -61.421, 65.053, -0.862, 86.354, 47.138]
  MoveL 484 to (129.11, 239.58, 0) mm, rotated rx 180 ry 0 rz -39.83 deg; joints [47.074, -61.451, 65.098, -0.862, 86.34, 47.125]
  MoveL 485 to (128.85, 239.22, 0) mm, rotated rx 180 ry 0 rz -39.83 deg; joints [47.061, -61.482, 65.144, -0.862, 86.325, 47.113]
  MoveL 486 to (128.59, 238.87, 0) mm, rotated rx 180 ry 0 rz -39.83 deg; joints [47.048, -61.513, 65.189, -0.862, 86.31, 47.1]
  MoveL 487 to (128.59, 238.87, 0) mm, rotated rx 180 ry 0 rz -39.83 deg; joints [47.048, -61.513, 65.189, -0.862, 86.31, 47.1]
  MoveL 488 to (128.36, 239.24, 0) mm, rotated rx 180 ry 0 rz -39.83 deg; joints [47.038, -61.478, 65.138, -0.862, 86.327, 47.09]
  MoveL 489 to (128.14, 239.61, 0) mm, rotated rx 180 ry 0 rz -39.83 deg; joints [47.029, -61.444, 65.086, -0.862, 86.344, 47.081]
  MoveL 490 to (127.93, 240, 0) mm, rotated rx 180 ry 0 rz -39.83 deg; joints [47.02, -61.408, 65.032, -0.862, 86.362, 47.072]
  MoveL 491 to (127.75, 240.39, 0) mm, rotated rx 180 ry 0 rz -39.83 deg; joints [47.013, -61.371, 64.978, -0.862, 86.38, 47.064]
  MoveL 492 to (127.63, 240.72, 0) mm, rotated rx 180 ry 0 rz -39.83 deg; joints [47.009, -61.342, 64.933, -0.862, 86.394, 47.06]
  MoveL 493 to (127.54, 241.05, 0) mm, rotated rx -180 ry 0 rz -39.83 deg; joints [47.005, -61.311, 64.888, -0.862, 86.409, 47.056]
  MoveL 494 to (127.48, 241.38, 0) mm, rotated rx -180 ry 0 rz -39.83 deg; joints [47.003, -61.281, 64.842, -0.862, 86.424, 47.054]
  MoveL 495 to (127.46, 241.72, 0) mm, rotated rx 180 ry 0 rz -39.83 deg; joints [47.003, -61.25, 64.797, -0.862, 86.439, 47.054]
  MoveL 496 to (127.48, 242.07, 0) mm, rotated rx 180 ry 0 rz -39.83 deg; joints [47.005, -61.219, 64.751, -0.862, 86.454, 47.055]
  MoveL 497 to (127.53, 242.41, 0) mm, rotated rx 180 ry 0 rz -39.83 deg; joints [47.008, -61.188, 64.705, -0.862, 86.469, 47.058]
  MoveL 498 to (127.6, 242.75, 0) mm, rotated rx 180 ry 0 rz -39.83 deg; joints [47.013, -61.158, 64.659, -0.862, 86.484, 47.062]
  MoveL 499 to (127.68, 243.09, 0) mm, rotated rx 180 ry 0 rz -39.83 deg; joints [47.017, -61.127, 64.614, -0.862, 86.499, 47.066]
  MoveL 500 to (127.71, 243.26, 0) mm, rotated rx 180 ry 0 rz -39.83 deg; joints [47.019, -61.112, 64.591, -0.862, 86.507, 47.068]
  MoveL 501 to (127.74, 243.43, 0) mm, rotated rx -180 ry 0 rz -39.83 deg; joints [47.02, -61.097, 64.569, -0.862, 86.514, 47.07]
  MoveL 502 to (127.77, 243.6, 0) mm, rotated rx -180 ry 0 rz -39.83 deg; joints [47.022, -61.082, 64.546, -0.862, 86.522, 47.071]
  MoveL 503 to (127.8, 243.77, 0) mm, rotated rx 180 ry 0 rz -39.83 deg; joints [47.024, -61.067, 64.523, -0.862, 86.529, 47.073]
  MoveL 504 to (127.8, 243.77, 0) mm, rotated rx 180 ry 0 rz -39.83 deg; joints [47.024, -61.067, 64.523, -0.862, 86.529, 47.073]
  MoveL 505 to (127.27, 243.44, 0) mm, rotated rx 180 ry 0 rz -39.83 deg; joints [46.999, -61.094, 64.563, -0.862, 86.516, 47.048]
  MoveL 506 to (126.75, 243.11, 0) mm, rotated rx -180 ry 0 rz -39.83 deg; joints [46.975, -61.121, 64.604, -0.862, 86.503, 47.024]
  MoveL 507 to (126.25, 242.75, 0) mm, rotated rx 180 ry 0 rz -39.83 deg; joints [46.951, -61.151, 64.647, -0.862, 86.489, 47]
  MoveL 508 to (125.77, 242.37, 0) mm, rotated rx 180 ry 0 rz -39.83 deg; joints [46.928, -61.183, 64.695, -0.862, 86.473, 46.978]
  MoveL 509 to (125.3, 241.93, 0) mm, rotated rx -180 ry 0 rz -39.83 deg; joints [46.905, -61.22, 64.75, -0.862, 86.455, 46.955]
  MoveL 510 to (124.85, 241.46, 0) mm, rotated rx 180 ry 0 rz -39.83 deg; joints [46.884, -61.261, 64.809, -0.862, 86.436, 46.934]
  MoveL 511 to (124.41, 240.98, 0) mm, rotated rx 180 ry 0 rz -39.83 deg; joints [46.862, -61.302, 64.87, -0.862, 86.416, 46.913]
  MoveL 512 to (123.98, 240.49, 0) mm, rotated rx 180 ry 0 rz -39.83 deg; joints [46.841, -61.344, 64.932, -0.862, 86.395, 46.892]
  MoveL 513 to (123.54, 240, 0) mm, rotated rx 180 ry 0 rz -39.83 deg; joints [46.82, -61.386, 64.994, -0.862, 86.375, 46.871]
  MoveL 514 to (123.09, 239.51, 0) mm, rotated rx 180 ry 0 rz -39.83 deg; joints [46.798, -61.427, 65.055, -0.862, 86.355, 46.85]
  MoveL 515 to (122.64, 239.04, 0) mm, rotated rx 180 ry 0 rz -39.83 deg; joints [46.776, -61.468, 65.115, -0.862, 86.336, 46.828]
  MoveL 516 to (122.17, 238.56, 0) mm, rotated rx 180 ry 0 rz -39.83 deg; joints [46.754, -61.508, 65.174, -0.862, 86.316, 46.806]
  MoveL 517 to (121.8, 238.18, 0) mm, rotated rx 180 ry 0 rz -39.83 deg; joints [46.735, -61.541, 65.222, -0.862, 86.301, 46.788]
  MoveL 518 to (121.43, 237.79, 0) mm, rotated rx 180 ry 0 rz -39.83 deg; joints [46.717, -61.574, 65.271, -0.862, 86.285, 46.77]
  MoveL 519 to (121.08, 237.39, 0) mm, rotated rx 180 ry 0 rz -39.83 deg; joints [46.7, -61.608, 65.321, -0.862, 86.268, 46.753]
  MoveL 520 to (120.75, 236.97, 0) mm, rotated rx 180 ry 0 rz -39.83 deg; joints [46.684, -61.644, 65.374, -0.862, 86.251, 46.737]
  MoveL 521 to (120.48, 236.58, 0) mm, rotated rx 180 ry 0 rz -39.83 deg; joints [46.671, -61.678, 65.424, -0.862, 86.235, 46.724]
  MoveL 522 to (120.24, 236.17, 0) mm, rotated rx 180 ry 0 rz -39.83 deg; joints [46.658, -61.713, 65.476, -0.862, 86.218, 46.712]
  MoveL 523 to (120.01, 235.75, 0) mm, rotated rx 180 ry 0 rz -39.83 deg; joints [46.647, -61.749, 65.529, -0.862, 86.201, 46.7]
  MoveL 524 to (119.78, 235.33, 0) mm, rotated rx 180 ry 0 rz -39.83 deg; joints [46.635, -61.786, 65.583, -0.862, 86.183, 46.689]
  MoveL 525 to (119.78, 235.33, 0) mm, rotated rx 180 ry 0 rz -39.83 deg; joints [46.635, -61.786, 65.583, -0.862, 86.183, 46.689]
  MoveL 526 to (119.53, 235.66, 0) mm, rotated rx 180 ry 0 rz -39.83 deg; joints [46.625, -61.755, 65.537, -0.862, 86.198, 46.678]
  MoveL 527 to (119.29, 236, 0) mm, rotated rx 180 ry 0 rz -39.83 deg; joints [46.614, -61.723, 65.49, -0.862, 86.214, 46.668]
  MoveL 528 to (119.06, 236.35, 0) mm, rotated rx 180 ry 0 rz -39.83 deg; joints [46.605, -61.691, 65.441, -0.862, 86.229, 46.658]
  MoveL 529 to (118.87, 236.71, 0) mm, rotated rx 180 ry 0 rz -39.83 deg; joints [46.597, -61.657, 65.391, -0.862, 86.246, 46.65]
  MoveL 530 to (118.71, 237.08, 0) mm, rotated rx -180 ry 0 rz -39.83 deg; joints [46.591, -61.623, 65.34, -0.862, 86.263, 46.644]
  MoveL 531 to (118.59, 237.47, 0) mm, rotated rx -180 ry 0 rz -39.83 deg; joints [46.587, -61.588, 65.288, -0.862, 86.28, 46.639]
  MoveL 532 to (118.51, 237.86, 0) mm, rotated rx 180 ry 0 rz -39.83 deg; joints [46.584, -61.552, 65.234, -0.862, 86.297, 46.636]
  MoveL 533 to (118.46, 238.26, 0) mm, rotated rx 180 ry 0 rz -39.83 deg; joints [46.583, -61.516, 65.18, -0.862, 86.315, 46.635]
  MoveL 534 to (118.44, 238.47, 0) mm, rotated rx 180 ry 0 rz -39.83 deg; joints [46.583, -61.496, 65.152, -0.862, 86.324, 46.635]
  MoveL 535 to (118.44, 238.69, 0) mm, rotated rx 180 ry 0 rz -39.83 deg; joints [46.583, -61.477, 65.123, -0.862, 86.334, 46.635]
  MoveL 536 to (118.43, 238.9, 0) mm, rotated rx 180 ry 0 rz -39.83 deg; joints [46.584, -61.458, 65.095, -0.862, 86.343, 46.635]
  MoveL 537 to (118.43, 239.11, 0) mm, rotated rx -180 ry 0 rz -39.83 deg; joints [46.584, -61.439, 65.066, -0.862, 86.352, 46.636]
  MoveL 538 to (118.43, 239.11, 0) mm, rotated rx -180 ry 0 rz -39.83 deg; joints [46.584, -61.439, 65.066, -0.862, 86.352, 46.636]
  MoveL 539 to (118.04, 238.78, 0) mm, rotated rx -180 ry 0 rz -39.83 deg; joints [46.565, -61.467, 65.107, -0.862, 86.339, 46.617]
  MoveL 540 to (117.66, 238.44, 0) mm, rotated rx -180 ry 0 rz -39.83 deg; joints [46.547, -61.495, 65.148, -0.862, 86.326, 46.599]
  MoveL 541 to (117.28, 238.1, 0) mm, rotated rx 180 ry 0 rz -39.83 deg; joints [46.528, -61.523, 65.19, -0.862, 86.312, 46.58]
  MoveL 542 to (116.9, 237.75, 0) mm, rotated rx 180 ry 0 rz -39.83 deg; joints [46.51, -61.553, 65.233, -0.862, 86.298, 46.563]
  MoveL 543 to (116.06, 236.85, 0) mm, rotated rx 180 ry 0 rz -39.83 deg; joints [46.469, -61.629, 65.345, -0.862, 86.261, 46.522]
  MoveL 544 to (115.27, 235.89, 0) mm, rotated rx 180 ry 0 rz -39.83 deg; joints [46.43, -61.711, 65.466, -0.862, 86.222, 46.483]
  MoveL 545 to (114.53, 234.89, 0) mm, rotated rx 180 ry 0 rz -39.83 deg; joints [46.393, -61.796, 65.591, -0.862, 86.181, 46.447]
  MoveL 546 to (113.82, 233.87, 0) mm, rotated rx 180 ry 0 rz -39.83 deg; joints [46.357, -61.884, 65.721, -0.862, 86.14, 46.412]
  MoveL 547 to (113.25, 233.01, 0) mm, rotated rx 180 ry 0 rz -39.83 deg; joints [46.329, -61.957, 65.828, -0.862, 86.105, 46.384]
  MoveL 548 to (112.69, 232.15, 0) mm, rotated rx 180 ry 0 rz -39.83 deg; joints [46.3, -62.031, 65.937, -0.862, 86.07, 46.356]
  MoveL 549 to (112.15, 231.28, 0) mm, rotated rx 180 ry 0 rz -39.83 deg; joints [46.273, -62.106, 66.046, -0.862, 86.034, 46.329]
  MoveL 550 to (111.63, 230.39, 0) mm, rotated rx 180 ry 0 rz -39.83 deg; joints [46.246, -62.182, 66.158, -0.862, 85.998, 46.303]
  MoveL 551 to (111.15, 229.52, 0) mm, rotated rx 180 ry 0 rz -39.83 deg; joints [46.221, -62.257, 66.268, -0.862, 85.963, 46.279]
  MoveL 552 to (110.7, 228.63, 0) mm, rotated rx 180 ry 0 rz -39.83 deg; joints [46.198, -62.333, 66.38, -0.862, 85.927, 46.255]
  MoveL 553 to (110.26, 227.73, 0) mm, rotated rx -180 ry 0 rz -39.83 deg; joints [46.175, -62.411, 66.493, -0.862, 85.891, 46.233]
  MoveL 554 to (109.85, 226.82, 0) mm, rotated rx 180 ry 0 rz -39.83 deg; joints [46.153, -62.489, 66.608, -0.862, 85.854, 46.212]
  MoveL 555 to (109.43, 225.85, 0) mm, rotated rx -180 ry 0 rz -39.83 deg; joints [46.13, -62.573, 66.732, -0.862, 85.814, 46.19]
  MoveL 556 to (109.05, 224.86, 0) mm, rotated rx 180 ry 0 rz -39.83 deg; joints [46.109, -62.659, 66.857, -0.863, 85.774, 46.169]
  MoveL 557 to (108.69, 223.87, 0) mm, rotated rx 180 ry 0 rz -39.83 deg; joints [46.089, -62.745, 66.983, -0.863, 85.734, 46.15]
  MoveL 558 to (108.36, 222.86, 0) mm, rotated rx 180 ry 0 rz -39.83 deg; joints [46.071, -62.832, 67.11, -0.863, 85.694, 46.132]
  MoveL 559 to (108.07, 221.88, 0) mm, rotated rx 180 ry 0 rz -39.83 deg; joints [46.054, -62.917, 67.234, -0.863, 85.654, 46.116]
  MoveL 560 to (107.82, 220.89, 0) mm, rotated rx 180 ry 0 rz -39.83 deg; joints [46.04, -63.003, 67.36, -0.863, 85.614, 46.102]
  MoveL 561 to (107.62, 219.9, 0) mm, rotated rx 180 ry 0 rz -39.83 deg; joints [46.027, -63.09, 67.487, -0.863, 85.574, 46.09]
  MoveL 562 to (107.47, 218.89, 0) mm, rotated rx 180 ry 0 rz -39.83 deg; joints [46.016, -63.178, 67.615, -0.863, 85.534, 46.08]
  MoveL 563 to (107.39, 218.2, 0) mm, rotated rx 180 ry 0 rz -39.83 deg; joints [46.011, -63.238, 67.703, -0.863, 85.506, 46.075]
  MoveL 564 to (107.35, 217.51, 0) mm, rotated rx -180 ry 0 rz -39.83 deg; joints [46.006, -63.299, 67.792, -0.863, 85.478, 46.071]
  MoveL 565 to (107.34, 216.81, 0) mm, rotated rx 180 ry 0 rz -39.83 deg; joints [46.004, -63.361, 67.882, -0.863, 85.45, 46.069]
  MoveL 566 to (107.37, 216.11, 0) mm, rotated rx 180 ry 0 rz -39.83 deg; joints [46.002, -63.422, 67.971, -0.863, 85.422, 46.068]
  MoveL 567 to (107.45, 215.21, 0) mm, rotated rx -180 ry 0 rz -39.83 deg; joints [46.003, -63.503, 68.089, -0.863, 85.385, 46.069]
  MoveL 568 to (107.59, 214.31, 0) mm, rotated rx 180 ry 0 rz -39.83 deg; joints [46.006, -63.583, 68.205, -0.863, 85.348, 46.073]
  MoveL 569 to (107.79, 213.42, 0) mm, rotated rx -180 ry 0 rz -39.83 deg; joints [46.013, -63.662, 68.321, -0.863, 85.312, 46.08]
  MoveL 570 to (108.06, 212.54, 0) mm, rotated rx -180 ry 0 rz -39.83 deg; joints [46.023, -63.741, 68.435, -0.863, 85.276, 46.09]
  MoveL 571 to (108.37, 211.76, 0) mm, rotated rx 180 ry 0 rz -39.83 deg; joints [46.034, -63.812, 68.539, -0.863, 85.244, 46.102]
  MoveL 572 to (108.74, 210.99, 0) mm, rotated rx 180 ry 0 rz -39.83 deg; joints [46.049, -63.881, 68.64, -0.863, 85.213, 46.118]
  MoveL 573 to (109.17, 210.26, 0) mm, rotated rx 180 ry 0 rz -39.83 deg; joints [46.066, -63.948, 68.738, -0.863, 85.182, 46.135]
  MoveL 574 to (109.65, 209.57, 0) mm, rotated rx -180 ry 0 rz -39.83 deg; joints [46.087, -64.011, 68.83, -0.863, 85.153, 46.156]
  MoveL 575 to (110.23, 208.87, 0) mm, rotated rx 180 ry 0 rz -39.83 deg; joints [46.112, -64.076, 68.924, -0.863, 85.124, 46.182]
  MoveL 576 to (110.87, 208.22, 0) mm, rotated rx 180 ry 0 rz -39.83 deg; joints [46.139, -64.137, 69.014, -0.863, 85.097, 46.21]
  MoveL 577 to (111.54, 207.6, 0) mm, rotated rx 180 ry 0 rz -39.83 deg; joints [46.169, -64.196, 69.099, -0.863, 85.07, 46.239]
  MoveL 578 to (112.23, 206.99, 0) mm, rotated rx -180 ry 0 rz -39.83 deg; joints [46.199, -64.253, 69.182, -0.863, 85.044, 46.27]
  MoveL 579 to (112.73, 206.56, 0) mm, rotated rx 180 ry 0 rz -39.83 deg; joints [46.221, -64.293, 69.241, -0.863, 85.026, 46.292]
  MoveL 580 to (113.24, 206.15, 0) mm, rotated rx -180 ry 0 rz -39.83 deg; joints [46.244, -64.332, 69.298, -0.864, 85.008, 46.315]
  MoveL 581 to (113.77, 205.76, 0) mm, rotated rx -180 ry 0 rz -39.83 deg; joints [46.267, -64.369, 69.352, -0.864, 84.992, 46.339]
  MoveL 582 to (114.31, 205.4, 0) mm, rotated rx 180 ry 0 rz -39.83 deg; joints [46.291, -64.403, 69.403, -0.864, 84.976, 46.364]
  MoveL 583 to (114.65, 205.21, 0) mm, rotated rx 180 ry 0 rz -39.83 deg; joints [46.307, -64.422, 69.43, -0.864, 84.968, 46.379]
  MoveL 584 to (114.99, 205.03, 0) mm, rotated rx -180 ry 0 rz -39.83 deg; joints [46.322, -64.44, 69.456, -0.864, 84.96, 46.395]
  MoveL 585 to (115.34, 204.86, 0) mm, rotated rx 180 ry 0 rz -39.83 deg; joints [46.338, -64.457, 69.481, -0.864, 84.952, 46.411]
  MoveL 586 to (115.69, 204.69, 0) mm, rotated rx -180 ry 0 rz -39.83 deg; joints [46.354, -64.474, 69.506, -0.864, 84.944, 46.427]
  MoveL 587 to (115.69, 204.69, 0) mm, rotated rx -180 ry 0 rz -39.83 deg; joints [46.354, -64.474, 69.506, -0.864, 84.944, 46.427]
  MoveL 588 to (126.36, 212.69, 0) mm, rotated rx 180 ry 0 rz -39.83 deg; joints [46.877, -63.829, 68.587, -0.863, 85.226, 46.945]
  MoveL 589 to (137.74, 219.57, 0) mm, rotated rx 180 ry 0 rz -39.83 deg; joints [47.424, -63.274, 67.794, -0.863, 85.472, 47.489]
  MoveL 590 to (149.76, 225.28, 0) mm, rotated rx 180 ry 0 rz -39.83 deg; joints [47.993, -62.812, 67.135, -0.863, 85.678, 48.055]
  MoveL 591 to (162.32, 229.76, 0) mm, rotated rx -180 ry 0 rz -39.83 deg; joints [48.581, -62.448, 66.616, -0.863, 85.841, 48.64]
  MoveL 592 to (162.32, 229.76, 0) mm, rotated rx -180 ry 0 rz -39.83 deg; joints [48.581, -62.448, 66.616, -0.863, 85.841, 48.64]
  MoveL 593 to (150.72, 223.79, 0) mm, rotated rx 180 ry 0 rz -39.83 deg; joints [48.035, -62.948, 67.334, -0.863, 85.615, 48.098]
  MoveL 594 to (139.67, 216.89, 0) mm, rotated rx 180 ry 0 rz -39.83 deg; joints [47.508, -63.518, 68.153, -0.863, 85.359, 47.574]
  MoveL 595 to (129.23, 209.1, 0) mm, rotated rx 180 ry 0 rz -39.83 deg; joints [47.001, -64.158, 69.067, -0.864, 85.077, 47.072]
  MoveL 596 to (119.45, 200.46, 0) mm, rotated rx 180 ry 0 rz -39.83 deg; joints [46.518, -64.863, 70.07, -0.864, 84.772, 46.593]
  Establecer velocidad (1000.0 mm/s)
  MoveL 597 to (119.45, 200.46, 0) mm, rotated rx 180 ry 0 rz -39.83 deg; joints [46.518, -64.863, 70.07, -0.864, 84.772, 46.593]
  MoveL 598 to (119.45, 200.46, 20) mm, rotated rx 180 ry 0 rz -39.83 deg; joints [46.532, -65.091, 68.674, -0.862, 86.395, 46.583]
